C01778=1013.630,227.704,-135.004,168.137,54.282,160.252
C01779=1013.625,227.455,-134.979,168.132,54.292,160.253
C01780=1013.620,227.206,-134.953,168.128,54.302,160.254
C01781=1013.615,226.958,-134.928,168.123,54.312,160.255
C01782=1013.611,226.709,-134.903,168.118,54.322,160.256
C01783=1013.604,226.460,-134.878,168.113,54.331,160.257
C01784=1013.600,226.211,-134.853,168.109,54.341,160.258
C01785=1013.595,225.963,-134.827,168.104,54.351,160.260
C01786=1013.590,225.714,-134.803,168.099,54.361,160.261
C01787=1013.584,225.465,-134.777,168.094,54.371,160.262
C01788=1013.579,225.217,-134.753,168.090,54.381,160.263
C01789=1013.574,224.968,-134.727,168.085,54.390,160.264
C01790=1013.565,224.568,-134.687,168.077,54.407,160.266
C01791=1013.557,224.167,-134.648,168.070,54.423,160.268
C01792=1013.549,223.766,-134.607,168.062,54.439,160.269
C01793=1013.541,223.365,-134.567,168.054,54.455,160.271
C01794=1013.535,223.116,-134.543,168.050,54.466,160.272
C01795=1013.530,222.868,-134.517,168.045,54.475,160.273
C01796=1013.524,222.619,-134.492,168.040,54.485,160.274
C01797=1013.520,222.370,-134.467,168.036,54.495,160.276
C01798=1013.515,222.122,-134.442,168.031,54.506,160.277
C01799=1013.510,221.873,-134.418,168.026,54.516,160.278
C01800=1013.505,221.624,-134.393,168.021,54.526,160.279
C01801=1013.499,221.375,-134.368,168.017,54.536,160.280
C01802=1013.494,221.127,-134.343,168.012,54.546,160.281
C01803=1013.489,220.878,-134.318,168.007,54.556,160.282
C01804=1013.485,220.629,-134.294,168.003,54.566,160.283
C01805=1013.479,220.381,-134.269,167.997,54.577,160.285
C01806=1013.475,220.132,-134.244,167.993,54.587,160.286
C01807=1013.469,219.883,-134.219,167.989,54.597,160.287
C01808=1013.464,219.634,-134.194,167.984,54.607,160.288
C01809=1013.459,219.386,-134.170,167.979,54.617,160.289
C01810=1013.452,219.034,-134.135,167.973,54.632,160.291
C01811=1013.444,218.683,-134.100,167.966,54.646,160.293
C01812=1013.437,218.332,-134.066,167.959,54.661,160.294
C01813=1013.431,217.981,-134.030,167.953,54.675,160.296
C01814=1013.425,217.732,-134.006,167.949,54.686,160.297
C01815=1013.421,217.483,-133.981,167.943,54.696,160.298
C01816=1013.415,217.235,-133.957,167.939,54.706,160.299
C01817=1013.410,216.986,-133.933,167.935,54.717,160.301
C01818=1013.405,216.737,-133.908,167.929,54.727,160.302
C01819=1013.400,216.489,-133.884,167.925,54.738,160.303
C01820=1013.395,216.240,-133.859,167.920,54.748,160.304
C01821=1013.390,215.991,-133.835,167.915,54.759,160.305
C01822=1013.385,215.742,-133.811,167.911,54.770,160.307
C01823=1013.379,215.494,-133.787,167.906,54.779,160.308
C01824=1013.375,215.245,-133.762,167.901,54.790,160.309
C01825=1013.370,214.996,-133.738,167.897,54.801,160.310
C01826=1013.364,214.747,-133.714,167.892,54.811,160.311
C01827=1013.359,214.499,-133.690,167.887,54.822,160.313
C01828=1013.354,214.250,-133.666,167.883,54.833,160.314
C01829=1013.349,214.001,-133.641,167.879,54.843,160.315
C01830=1013.344,213.752,-133.617,167.873,54.854,160.316
C01831=1013.339,213.504,-133.593,167.869,54.864,160.318
C01832=1013.334,213.254,-133.569,167.864,54.875,160.319
C01833=1013.329,213.006,-133.545,167.860,54.886,160.320
C01834=1013.324,212.757,-133.520,167.855,54.896,160.321
C01835=1013.319,212.508,-133.496,167.850,54.907,160.322
C01836=1013.314,212.259,-133.472,167.846,54.918,160.324
C01837=1013.308,212.010,-133.448,167.841,54.929,160.325
C01838=1013.304,211.762,-133.423,167.837,54.939,160.326
C01839=1013.299,211.512,-133.400,167.832,54.949,160.327
C01840=1013.294,211.264,-133.376,167.827,54.960,160.329
C01841=1013.289,211.016,-133.351,167.823,54.971,160.330
C01842=1013.284,210.767,-133.328,167.818,54.982,160.331
C01843=1013.279,210.518,-133.303,167.814,54.993,160.332
C01844=1013.274,210.269,-133.279,167.809,55.003,160.334
C01845=1013.269,210.020,-133.255,167.804,55.014,160.335
C01846=1013.264,209.771,-133.231,167.800,55.024,160.336
C01847=1013.259,209.522,-133.207,167.795,55.035,160.337
C01848=1013.255,209.274,-133.183,167.791,55.046,160.339
C01849=1013.250,209.025,-133.159,167.785,55.057,160.340
C01850=1013.244,208.776,-133.135,167.781,55.068,160.341
C01851=1013.239,208.527,-133.112,167.776,55.079,160.342
C01852=1013.234,208.278,-133.087,167.772,55.090,160.344
C01853=1013.230,208.030,-133.064,167.767,55.101,160.345
C01854=1013.224,207.781,-133.040,167.763,55.111,160.346
C01855=1013.219,207.532,-133.016,167.758,55.122,160.347
C01856=1013.214,207.283,-132.993,167.754,55.133,160.349
C01857=1013.209,207.034,-132.969,167.749,55.144,160.350
C01858=1013.205,206.786,-132.945,167.745,55.156,160.352
C01859=1013.199,206.537,-132.921,167.740,55.167,160.353
C01860=1013.194,206.288,-132.898,167.735,55.178,160.354
C01861=1013.189,206.039,-132.874,167.731,55.188,160.355
C01862=1013.184,205.791,-132.851,167.726,55.200,160.357
C01863=1013.179,205.542,-132.827,167.722,55.210,160.358
C01864=1013.174,205.293,-132.804,167.717,55.221,160.359
C01865=1013.169,205.044,-132.780,167.713,55.233,160.361
C01866=1013.164,204.796,-132.756,167.708,55.244,160.362
C01867=1013.159,204.547,-132.733,167.703,55.255,160.363
C01868=1013.154,204.297,-132.709,167.699,55.266,160.365
C01869=1013.150,204.049,-132.686,167.695,55.278,160.366
C01870=1013.144,203.798,-132.662,167.690,55.289,160.367
C01871=1013.139,203.546,-132.638,167.685,55.300,160.368
C01872=1013.134,203.295,-132.616,167.681,55.311,160.370
C01873=1013.129,203.043,-132.592,167.676,55.322,160.371
C01874=1013.112,202.020,-132.502,167.137,55.220,160.221
C01875=1013.109,201.771,-132.481,167.133,55.232,160.223
C01876=1013.105,201.522,-132.458,167.127,55.245,160.224
C01877=1013.101,201.273,-132.438,167.123,55.257,160.226
C01878=1013.097,201.024,-132.415,167.119,55.269,160.227
C01879=1013.094,200.775,-132.394,167.114,55.282,160.229
C01880=1013.089,200.526,-132.372,167.109,55.294,160.230
C01881=1013.086,200.277,-132.351,167.105,55.306,160.232
C01882=1013.082,200.027,-132.329,167.100,55.318,160.233
C01883=1013.078,199.779,-132.307,167.094,55.331,160.234
C01884=1013.074,199.529,-132.286,167.090,55.343,160.236
C01885=1013.071,199.281,-132.264,167.086,55.355,160.237
C01886=1013.066,199.032,-132.242,167.082,55.368,160.239
C01887=1013.063,198.783,-132.221,167.076,55.380,160.240
C01888=1013.058,198.533,-132.200,167.072,55.393,160.242
C01889=1013.055,198.284,-132.178,167.067,55.405,160.243
C01890=1013.050,198.035,-132.157,167.063,55.417,160.245
C01891=1013.046,197.787,-132.136,167.058,55.429,160.246
C01892=1013.043,197.537,-132.114,167.053,55.442,160.247
C01893=1013.039,197.288,-132.093,167.049,55.454,160.249
C01894=1013.035,197.039,-132.073,167.044,55.467,160.250
C01895=1013.030,196.790,-132.051,167.039,55.479,160.252
C01896=1013.027,196.541,-132.030,167.035,55.492,160.253
C01897=1013.023,196.291,-132.009,167.031,55.504,160.255
C01898=1013.019,196.043,-131.988,167.025,55.517,160.256
C01899=1013.015,195.793,-131.966,167.021,55.529,160.258
C01900=1013.011,195.544,-131.946,167.017,55.541,160.259
C01901=1013.007,195.295,-131.925,167.013,55.554,160.261
C01902=1013.003,195.046,-131.904,167.007,55.566,160.262
C01903=1012.999,194.797,-131.882,167.003,55.579,160.264
C01904=1012.995,194.548,-131.861,166.998,55.591,160.265
C01905=1012.991,194.299,-131.840,166.994,55.603,160.266
C01906=1012.987,194.050,-131.820,166.990,55.615,160.268
C01907=1012.984,193.801,-131.798,166.984,55.628,160.269
C01908=1012.979,193.552,-131.777,166.980,55.640,160.271
C01909=1012.975,193.303,-131.756,166.976,55.652,160.272
C01910=1012.972,193.054,-131.735,166.972,55.665,160.274
C01911=1012.968,192.804,-131.714,166.967,55.677,160.275
C01912=1012.964,192.556,-131.693,166.963,55.690,160.277
C01913=1012.960,192.307,-131.672,166.959,55.702,160.278
C01914=1012.956,192.057,-131.650,166.955,55.714,160.280
C01915=1012.952,191.808,-131.630,166.949,55.727,160.281
C01916=1012.949,191.559,-131.610,166.945,55.739,160.282
C01917=1012.945,191.310,-131.589,166.941,55.751,160.284
C01918=1012.941,191.061,-131.567,166.936,55.763,160.285
C01919=1012.937,190.812,-131.546,166.932,55.776,160.287
C01920=1012.933,190.563,-131.525,166.928,55.788,160.288
C01921=1012.930,190.314,-131.504,166.923,55.800,160.290
C01922=1012.926,190.064,-131.484,166.919,55.813,160.291
C01923=1012.922,189.815,-131.463,166.915,55.825,160.293
C01924=1012.918,189.567,-131.442,166.911,55.837,160.294
C01925=1012.915,189.318,-131.421,166.906,55.849,160.296
C01926=1012.910,189.068,-131.400,166.902,55.861,160.297
C01927=1012.907,188.819,-131.379,166.898,55.874,160.299
C01928=1012.903,188.570,-131.359,166.893,55.886,160.300
C01929=1012.899,188.321,-131.337,166.889,55.898,160.302
C01930=1012.896,188.072,-131.317,166.885,55.911,160.303
C01931=1012.891,187.822,-131.296,166.880,55.923,160.305
C01932=1012.887,187.573,-131.275,166.876,55.935,160.306
C01933=1012.884,187.324,-131.254,166.872,55.948,160.308
C01934=1012.880,187.076,-131.233,166.867,55.960,160.309
C01935=1012.876,186.796,-131.210,166.863,55.973,160.311
C01936=1012.872,186.518,-131.186,166.858,55.987,160.312
C01937=1012.868,186.240,-131.164,166.854,56.001,160.314
C01938=1012.863,185.960,-131.140,166.849,56.014,160.315
C01939=1012.860,185.711,-131.120,166.845,56.026,160.317
C01940=1012.857,185.462,-131.099,166.840,56.038,160.319
C01941=1012.853,185.213,-131.079,166.836,56.051,160.320
C01942=1012.849,184.964,-131.058,166.832,56.063,160.322
C01943=1012.845,184.715,-131.037,166.829,56.075,160.323
C01944=1012.842,184.466,-131.016,166.824,56.087,160.324
C01945=1012.838,184.216,-130.995,166.820,56.099,160.326
C01946=1012.834,183.967,-130.974,166.816,56.112,160.328
C01947=1012.830,183.718,-130.954,166.811,56.124,160.329
C01948=1012.827,183.469,-130.933,166.807,56.136,160.330
C01949=1012.823,183.220,-130.913,166.804,56.148,160.332
C01950=1012.820,182.971,-130.892,166.799,56.160,160.333
C01951=1012.816,182.722,-130.872,166.795,56.172,160.335
C01952=1012.813,182.472,-130.851,166.791,56.184,160.336
C01953=1012.809,182.224,-130.830,166.788,56.196,160.338
C01954=1012.805,181.974,-130.810,166.783,56.208,160.339
C01955=1012.802,181.725,-130.789,166.779,56.220,160.341
C01956=1012.798,181.476,-130.768,166.774,56.232,160.342
C01957=1012.795,181.227,-130.748,166.772,56.245,160.344
C01958=1012.791,180.977,-130.728,166.767,56.257,160.345
C01959=1012.786,180.728,-130.708,166.763,56.270,160.347
C01960=1012.782,180.479,-130.688,166.759,56.282,160.348
C01961=1012.778,180.230,-130.668,166.755,56.294,160.350
C01962=1012.774,179.980,-130.648,166.751,56.307,160.351
C01963=1012.771,179.731,-130.628,166.746,56.319,160.353
C01964=1012.766,179.482,-130.609,166.742,56.331,160.354
C01965=1012.763,179.233,-130.589,166.738,56.344,160.356
C01966=1012.759,178.984,-130.569,166.735,56.355,160.357
C01967=1012.755,178.734,-130.549,166.731,56.368,160.359
C01968=1012.751,178.485,-130.529,166.727,56.380,160.360
C01969=1012.747,178.236,-130.509,166.722,56.392,160.362
C01970=1012.743,177.987,-130.489,166.719,56.405,160.363
C01971=1012.739,177.738,-130.469,166.715,56.417,160.365
C01972=1012.736,177.489,-130.449,166.711,56.429,160.366
C01973=1012.732,177.240,-130.429,166.707,56.441,160.368
C01974=1012.728,176.991,-130.410,166.703,56.454,160.369
C01975=1012.724,176.742,-130.390,166.699,56.466,160.371
C01976=1012.720,176.493,-130.370,166.695,56.478,160.372
C01977=1012.716,176.243,-130.350,166.692,56.491,160.374
C01978=1012.712,175.994,-130.331,166.687,56.503,160.375
C01979=1012.708,175.745,-130.311,166.683,56.515,160.377
C01980=1012.705,175.496,-130.291,166.680,56.527,160.378
C01981=1012.701,175.246,-130.272,166.676,56.540,160.380
C01982=1012.697,174.997,-130.252,166.672,56.552,160.382
C01983=1012.693,174.748,-130.232,166.668,56.563,160.383
C01984=1012.689,174.498,-130.212,166.664,56.576,160.384
C01985=1012.686,174.250,-130.193,166.660,56.588,160.386
C01986=1012.682,174.000,-130.173,166.657,56.600,160.388
C01987=1012.678,173.751,-130.153,166.653,56.612,160.389
C01988=1012.674,173.502,-130.134,166.649,56.624,160.391
C01989=1012.670,173.253,-130.114,166.645,56.636,160.392
C01990=1012.666,173.003,-130.094,166.641,56.648,160.394
C01991=1012.662,172.754,-130.074,166.638,56.660,160.395
C01992=1012.659,172.505,-130.055,166.634,56.673,160.397
C01993=1012.655,172.256,-130.036,166.630,56.685,160.398
C01994=1012.651,172.007,-130.016,166.627,56.697,160.400
C01995=1012.648,171.757,-129.995,166.622,56.709,160.401
C01996=1012.643,171.508,-129.976,166.619,56.721,160.403
C01997=1012.640,171.259,-129.956,166.615,56.733,160.404
C01998=1012.636,171.011,-129.937,166.611,56.745,160.406
C01999=1012.632,170.707,-129.913,166.607,56.760,160.408
C02000=1012.627,170.404,-129.889,166.602,56.775,160.409
C02001=1012.623,170.100,-129.865,166.598,56.789,160.411
C02002=1012.618,169.798,-129.841,166.593,56.804,160.413
C02003=1012.614,169.548,-129.822,166.590,56.816,160.415
C02004=1012.611,169.299,-129.802,166.586,56.828,160.416
C02005=1012.607,169.050,-129.783,166.582,56.840,160.418
C02006=1012.603,168.801,-129.763,166.578,56.852,160.419
C02007=1012.599,168.551,-129.744,166.575,56.864,160.421
C02008=1012.596,168.302,-129.724,166.571,56.876,160.422
C02009=1012.592,168.054,-129.705,166.568,56.888,160.424
C02010=1012.588,167.804,-129.685,166.565,56.899,160.425
C02011=1012.585,167.554,-129.666,166.560,56.912,160.427
C02012=1012.581,167.305,-129.646,166.557,56.923,160.428
C02013=1012.578,167.057,-129.626,166.553,56.936,160.430
C02014=1012.574,166.807,-129.608,166.550,56.947,160.431
C02015=1012.570,166.558,-129.588,166.547,56.959,160.433
C02016=1012.567,166.309,-129.568,166.543,56.971,160.434
C02017=1012.563,166.060,-129.548,166.539,56.983,160.436
C02018=1012.559,165.810,-129.529,166.536,56.995,160.437
C02019=1012.556,165.562,-129.510,166.532,57.007,160.439
C02020=1012.552,165.312,-129.491,166.529,57.019,160.440
C02021=1012.548,165.063,-129.471,166.525,57.030,160.442
C02022=1012.545,164.814,-129.451,166.521,57.042,160.443
C02023=1012.542,164.564,-129.432,166.518,57.054,160.445
C02024=1012.537,164.315,-129.413,166.515,57.066,160.446
C02025=1012.534,164.066,-129.393,166.512,57.078,160.448
C02026=1012.530,163.817,-129.374,166.508,57.090,160.449
C02027=1012.527,163.567,-129.354,166.504,57.101,160.451
C02028=1012.524,163.318,-129.335,166.501,57.113,160.452
C02029=1012.520,163.069,-129.316,166.498,57.125,160.454
C02030=1012.516,162.820,-129.296,166.494,57.137,160.455
C02031=1012.494,177.789,-130.860,166.672,56.580,160.387
C02032=1012.498,178.038,-130.880,166.675,56.568,160.386
C02033=1012.501,178.288,-130.900,166.679,56.556,160.384
C02034=1012.505,178.537,-130.920,166.683,56.543,160.383
C02035=1012.509,178.786,-130.939,166.687,56.531,160.381
C02036=1012.512,179.035,-130.959,166.692,56.519,160.380
C02037=1012.517,179.284,-130.978,166.695,56.507,160.378
C02038=1012.520,179.533,-130.998,166.699,56.494,160.377
C02039=1012.524,179.783,-131.018,166.703,56.482,160.375
C02040=1012.528,180.032,-131.038,166.707,56.470,160.374
C02041=1012.532,180.281,-131.058,166.711,56.457,160.372
C02042=1012.536,180.530,-131.078,166.715,56.445,160.371
C02043=1012.540,180.779,-131.098,166.719,56.433,160.369
C02044=1012.544,181.029,-131.118,166.722,56.421,160.368
C02045=1012.548,181.278,-131.137,166.727,56.409,160.366
C02046=1012.551,181.527,-131.157,166.731,56.396,160.365
C02047=1012.555,181.776,-131.179,166.736,56.384,160.363
C02048=1012.558,182.026,-131.199,166.739,56.373,160.362
C02049=1012.562,182.274,-131.219,166.743,56.361,160.360
C02050=1012.565,182.524,-131.240,166.747,56.348,160.359
C02051=1012.569,182.773,-131.261,166.751,56.336,160.357
C02052=1012.573,183.022,-131.281,166.756,56.323,160.356
C02053=1012.577,183.271,-131.302,166.759,56.312,160.354
C02054=1012.579,183.520,-131.322,166.763,56.300,160.353
C02055=1012.583,183.769,-131.343,166.768,56.288,160.352
C02056=1012.587,184.019,-131.363,166.772,56.275,160.350
C02057=1012.591,184.267,-131.384,166.776,56.263,160.349
C02058=1012.594,184.517,-131.405,166.779,56.251,160.347
C02059=1012.598,184.766,-131.425,166.784,56.239,160.346
C02060=1012.601,185.015,-131.445,166.788,56.227,160.344
C02061=1012.605,185.264,-131.466,166.792,56.214,160.343
C02062=1012.608,185.513,-131.487,166.796,56.202,160.341
C02063=1012.612,185.762,-131.508,166.801,56.190,160.340
C02064=1012.617,186.082,-131.534,166.806,56.175,160.338
C02065=1012.622,186.401,-131.561,166.811,56.159,160.336
C02066=1012.627,186.720,-131.587,166.817,56.143,160.334
C02067=1012.631,187.040,-131.614,166.821,56.127,160.332
C02068=1012.635,187.289,-131.635,166.826,56.115,160.331
C02069=1012.638,187.538,-131.655,166.830,56.103,160.329
C02070=1012.642,187.787,-131.676,166.834,56.091,160.328
C02071=1012.645,188.036,-131.697,166.838,56.079,160.326
C02072=1012.649,188.285,-131.717,166.843,56.067,160.325
C02073=1012.653,188.534,-131.738,166.847,56.054,160.323
C02074=1012.657,188.783,-131.759,166.851,56.042,160.322
C02075=1012.660,189.033,-131.780,166.855,56.030,160.320
C02076=1012.664,189.282,-131.801,166.860,56.018,160.319
C02077=1012.668,189.531,-131.821,166.864,56.005,160.317
C02078=1012.672,189.780,-131.842,166.868,55.993,160.316
C02079=1012.675,190.029,-131.863,166.872,55.980,160.314
C02080=1012.679,190.278,-131.884,166.877,55.968,160.313
C02081=1012.683,190.527,-131.904,166.881,55.956,160.312
C02082=1012.687,190.777,-131.925,166.885,55.943,160.310
C02083=1012.690,191.026,-131.946,166.889,55.931,160.309
C02084=1012.694,191.274,-131.967,166.895,55.919,160.307
C02085=1012.698,191.523,-131.988,166.899,55.906,160.306
C02086=1012.701,191.773,-132.008,166.903,55.894,160.304
C02087=1012.705,192.022,-132.030,166.907,55.881,160.303
C02088=1012.709,192.271,-132.050,166.912,55.869,160.301
C02089=1012.713,192.520,-132.071,166.916,55.857,160.300
C02090=1012.716,192.769,-132.093,166.920,55.845,160.298
C02091=1012.721,193.019,-132.113,166.925,55.833,160.297
C02092=1012.724,193.268,-132.134,166.930,55.820,160.295
C02093=1012.728,193.516,-132.155,166.934,55.808,160.294
C02094=1012.732,193.765,-132.176,166.938,55.795,160.292
C02095=1012.736,194.015,-132.197,166.943,55.783,160.291
C02096=1012.740,194.264,-132.218,166.947,55.771,160.290
C02097=1012.743,194.513,-132.239,166.952,55.758,160.288
C02098=1012.748,194.762,-132.260,166.957,55.746,160.287
C02099=1012.751,195.011,-132.280,166.961,55.733,160.285
C02100=1012.755,195.260,-132.301,166.965,55.721,160.284
C02101=1012.759,195.510,-132.323,166.969,55.708,160.282
C02102=1012.763,195.759,-132.344,166.975,55.696,160.281
C02103=1012.767,196.007,-132.365,166.979,55.683,160.279
C02104=1012.771,196.257,-132.386,166.983,55.671,160.278
C02105=1012.775,196.506,-132.407,166.987,55.659,160.276
C02106=1012.778,196.755,-132.428,166.993,55.646,160.275
C02107=1012.783,197.004,-132.449,166.997,55.634,160.273
C02108=1012.786,197.253,-132.470,167.002,55.622,160.272
C02109=1012.790,197.502,-132.491,167.007,55.609,160.271
C02110=1012.795,197.751,-132.512,167.011,55.597,160.269
C02111=1012.798,198.000,-132.533,167.015,55.584,160.268
C02112=1012.802,198.249,-132.554,167.020,55.571,160.266
C02113=1012.806,198.498,-132.576,167.025,55.559,160.265
C02114=1012.810,198.747,-132.596,167.029,55.546,160.263
C02115=1012.814,198.996,-132.619,167.035,55.534,160.262
C02116=1012.817,199.245,-132.640,167.039,55.522,160.261
C02117=1012.822,199.495,-132.661,167.043,55.510,160.259
C02118=1012.825,199.744,-132.683,167.048,55.498,160.258
C02119=1012.829,199.992,-132.705,167.053,55.485,160.256
C02120=1012.833,200.242,-132.726,167.057,55.473,160.255
C02121=1012.836,200.491,-132.747,167.061,55.460,160.253
C02122=1012.840,200.740,-132.770,167.067,55.448,160.252
C02123=1012.844,200.989,-132.791,167.071,55.435,160.250
C02124=1012.848,201.238,-132.812,167.076,55.423,160.249
C02125=1012.852,201.487,-132.834,167.081,55.411,160.248
C02126=1012.855,201.735,-132.855,167.086,55.398,160.246
C02127=1012.860,201.985,-132.878,167.090,55.386,160.245
C02128=1012.874,202.987,-132.965,167.632,55.486,160.396
C02129=1012.880,203.246,-132.989,167.637,55.475,160.395
C02130=1012.886,203.504,-133.013,167.643,55.463,160.393
C02131=1012.890,203.764,-133.037,167.647,55.451,160.392
C02132=1012.895,204.022,-133.061,167.652,55.439,160.391
C02133=1012.900,204.271,-133.085,167.655,55.428,160.389
C02134=1012.905,204.520,-133.108,167.661,55.417,160.388
C02135=1012.911,204.769,-133.131,167.666,55.406,160.387
C02136=1012.916,205.018,-133.155,167.669,55.395,160.385
C02137=1012.921,205.267,-133.178,167.674,55.384,160.384
C02138=1012.925,205.515,-133.202,167.679,55.372,160.383
C02139=1012.930,205.764,-133.226,167.683,55.362,160.381
C02140=1012.935,206.013,-133.249,167.688,55.351,160.380
C02141=1012.940,206.262,-133.272,167.693,55.339,160.379
C02142=1012.945,206.510,-133.297,167.697,55.329,160.378
C02143=1012.950,206.760,-133.320,167.702,55.318,160.376
C02144=1012.955,207.009,-133.344,167.706,55.307,160.375
C02145=1012.959,207.257,-133.367,167.711,55.296,160.374
C02146=1012.965,207.506,-133.391,167.716,55.285,160.373
C02147=1012.970,207.755,-133.415,167.720,55.273,160.371
C02148=1012.975,208.004,-133.438,167.725,55.262,160.370
C02149=1012.979,208.252,-133.462,167.729,55.251,160.368
C02150=1012.984,208.501,-133.486,167.734,55.240,160.367
C02151=1012.990,208.750,-133.510,167.738,55.229,160.366
C02152=1012.995,208.999,-133.533,167.743,55.219,160.365
C02153=1012.999,209.248,-133.557,167.747,55.208,160.364
C02154=1013.004,209.496,-133.581,167.753,55.197,160.362
C02155=1013.009,209.746,-133.604,167.757,55.187,160.361
C02156=1013.014,209.994,-133.629,167.762,55.175,160.360
C02157=1013.019,210.244,-133.653,167.766,55.165,160.358
C02158=1013.023,210.491,-133.677,167.771,55.154,160.357
C02159=1013.029,210.740,-133.701,167.775,55.143,160.356
C02160=1013.034,210.989,-133.724,167.780,55.133,160.355
C02161=1013.038,211.238,-133.749,167.784,55.122,160.354
C02162=1013.043,211.487,-133.773,167.790,55.111,160.352
C02163=1013.049,211.736,-133.797,167.794,55.100,160.351
C02164=1013.053,211.984,-133.820,167.799,55.089,160.350
C02165=1013.058,212.233,-133.844,167.803,55.079,160.349
C02166=1013.063,212.482,-133.869,167.808,55.068,160.348
C02167=1013.068,212.731,-133.893,167.812,55.057,160.346
C02168=1013.073,212.980,-133.917,167.816,55.047,160.345
C02169=1013.078,213.228,-133.941,167.822,55.036,160.344
C02170=1013.083,213.478,-133.966,167.826,55.026,160.343
C02171=1013.088,213.726,-133.990,167.831,55.015,160.341
C02172=1013.093,213.975,-134.014,167.835,55.004,160.340
C02173=1013.098,214.224,-134.038,167.841,54.994,160.339
C02174=1013.103,214.472,-134.061,167.845,54.983,160.338
C02175=1013.108,214.721,-134.086,167.849,54.972,160.336
C02176=1013.113,214.970,-134.111,167.854,54.961,160.335
C02177=1013.118,215.219,-134.134,167.859,54.951,160.334
C02178=1013.123,215.467,-134.158,167.864,54.940,160.333
C02179=1013.128,215.716,-134.183,167.868,54.930,160.331
C02180=1013.133,215.965,-134.207,167.873,54.920,160.330
C02181=1013.138,216.214,-134.231,167.878,54.909,160.329
C02182=1013.143,216.463,-134.255,167.883,54.899,160.328
C02183=1013.149,216.711,-134.280,167.888,54.888,160.327
C02184=1013.153,216.960,-134.304,167.892,54.877,160.326
C02185=1013.158,217.209,-134.329,167.896,54.867,160.324
C02186=1013.164,217.457,-134.353,167.902,54.856,160.323
C02187=1013.169,217.706,-134.377,167.906,54.846,160.322
C02188=1013.174,217.955,-134.402,167.910,54.835,160.321
C02189=1013.179,218.212,-134.427,167.915,54.824,160.320
C02190=1013.183,218.468,-134.453,167.920,54.814,160.319
C02191=1013.189,218.726,-134.478,167.925,54.803,160.317
C02192=1013.195,218.982,-134.503,167.930,54.792,160.316
C02193=1013.199,219.231,-134.528,167.935,54.782,160.315
C02194=1013.205,219.480,-134.552,167.939,54.772,160.314
C02195=1013.209,219.729,-134.577,167.944,54.762,160.313
C02196=1013.214,219.977,-134.601,167.949,54.752,160.312
C02197=1013.219,220.226,-134.626,167.954,54.741,160.310
C02198=1013.224,220.475,-134.652,167.958,54.731,160.309
C02199=1013.229,220.723,-134.676,167.963,54.721,160.308
C02200=1013.234,220.972,-134.701,167.967,54.711,160.307
C02201=1013.240,221.221,-134.725,167.973,54.700,160.306
C02202=1013.244,221.470,-134.750,167.977,54.690,160.305
C02203=1013.249,221.719,-134.775,167.982,54.680,160.303
C02204=1013.254,221.968,-134.799,167.986,54.670,160.302
C02205=1013.260,222.216,-134.824,167.992,54.660,160.301
C02206=1013.264,222.465,-134.849,167.997,54.650,160.300
C02207=1013.269,222.713,-134.873,168.001,54.639,160.299
C02208=1013.275,222.963,-134.899,168.005,54.629,160.298
C02209=1013.280,223.211,-134.924,168.010,54.619,160.297
C02210=1013.285,223.460,-134.948,168.016,54.609,160.296
C02211=1013.290,223.708,-134.973,168.020,54.599,160.295
C02212=1013.295,223.957,-134.998,168.025,54.589,160.293
C02213=1013.301,224.206,-135.023,168.029,54.579,160.292
C02214=1013.305,224.455,-135.048,168.034,54.569,160.291
C02215=1013.311,224.703,-135.072,168.040,54.559,160.290
C02216=1013.316,224.952,-135.098,168.044,54.548,160.289
C02217=1013.321,225.200,-135.122,168.049,54.538,160.288
C02218=1013.326,225.450,-135.147,168.053,54.528,160.287
C02219=1013.332,225.698,-135.172,168.058,54.518,160.286
C02220=1013.336,225.947,-135.197,168.063,54.509,160.285
C02221=1013.341,226.195,-135.222,168.067,54.499,160.284
C02222=1013.346,226.443,-135.247,168.072,54.489,160.282
C02223=1013.352,226.692,-135.273,168.078,54.479,160.282
C02224=1013.356,226.941,-135.297,168.083,54.469,160.280
C02225=1013.361,227.190,-135.323,168.087,54.459,160.279
C02226=1013.366,227.439,-135.348,168.092,54.449,160.278
C02227=1013.372,227.687,-135.373,168.097,54.439,160.277
C02228=1013.377,227.935,-135.399,168.101,54.429,160.276
C02229=1013.381,228.184,-135.424,168.106,54.420,160.275
C02230=1013.387,228.433,-135.450,168.111,54.410,160.274
C02231=1013.392,228.682,-135.474,168.116,54.400,160.273
C02232=1013.397,228.930,-135.499,168.120,54.390,160.272
C02233=1013.403,229.179,-135.525,168.125,54.380,160.271
C02234=1013.407,229.428,-135.550,168.130,54.370,160.270
C02235=1013.412,229.676,-135.576,168.135,54.361,160.269
C02236=1013.417,229.925,-135.602,168.140,54.351,160.268
C02237=1013.422,230.174,-135.627,168.144,54.342,160.267
C02238=1013.428,230.422,-135.652,168.149,54.332,160.266
C02239=1013.433,230.671,-135.677,168.154,54.322,160.264
C02240=1013.438,230.919,-135.703,168.159,54.313,160.264
C02241=1013.443,231.168,-135.729,168.164,54.303,160.263
C02242=1013.448,231.417,-135.754,168.169,54.293,160.261
C02243=1013.453,231.666,-135.779,168.173,54.283,160.260
C02244=1013.458,231.915,-135.805,168.179,54.274,160.260
C02245=1013.463,232.163,-135.831,168.183,54.264,160.258
C02246=1013.469,232.412,-135.857,168.188,54.255,160.257
C02247=1013.473,232.660,-135.882,168.193,54.245,160.257
C02248=1013.478,232.908,-135.908,168.198,54.236,160.255
C02249=1013.485,233.227,-135.940,168.204,54.224,160.254
C02250=1013.492,233.548,-135.974,168.211,54.211,160.253
C02251=1013.499,233.866,-136.007,168.217,54.199,160.252
C02252=1013.505,234.185,-136.039,168.223,54.187,160.250
C02253=1013.510,234.433,-136.065,168.227,54.178,160.249
C02254=1013.516,234.682,-136.090,168.232,54.168,160.248
C02255=1013.521,234.931,-136.116,168.237,54.159,160.247
C02256=1013.526,235.180,-136.142,168.242,54.149,160.246
C02257=1013.531,235.428,-136.168,168.247,54.140,160.245
C02258=1013.536,235.677,-136.193,168.252,54.130,160.244
C02259=1013.541,235.925,-136.219,168.257,54.121,160.243
C02260=1013.547,236.174,-136.245,168.262,54.111,160.242
C02261=1013.552,236.422,-136.271,168.267,54.102,160.242
C02262=1013.557,236.671,-136.296,168.272,54.092,160.240
C02263=1013.562,236.919,-136.323,168.276,54.084,160.239
C02264=1013.568,237.168,-136.349,168.281,54.074,160.238
C02265=1013.573,237.417,-136.375,168.286,54.065,160.238
C02266=1013.578,237.665,-136.400,168.291,54.055,160.236
C02267=1013.584,237.914,-136.426,168.297,54.046,160.236
C02268=1013.588,238.163,-136.452,168.301,54.036,160.235
C02269=1013.594,238.412,-136.478,168.307,54.027,160.234
C02270=1013.598,238.659,-136.505,168.311,54.018,160.233
C02271=1013.604,238.908,-136.530,168.316,54.009,160.232
C02272=1013.609,239.157,-136.556,168.321,54.000,160.231
C02273=1013.614,239.405,-136.583,168.326,53.990,160.230
C02274=1013.619,239.654,-136.609,168.331,53.982,160.229
C02275=1013.625,239.903,-136.635,168.335,53.972,160.228
C02276=1013.630,240.151,-136.661,168.341,53.963,160.227
C02277=1013.634,240.364,-136.685,168.344,53.955,160.226
C02278=1013.639,240.578,-136.706,168.349,53.947,160.226
C02279=1013.643,240.791,-136.729,168.353,53.940,160.225
C02280=1013.648,241.004,-136.752,168.358,53.932,160.224
C02281=1013.652,241.218,-136.774,168.361,53.924,160.223
C02282=1013.656,241.430,-136.797,168.366,53.916,160.222
C02283=1013.661,241.644,-136.819,168.370,53.909,160.222
C02284=1013.666,241.857,-136.842,168.375,53.901,160.221
C02285=1013.670,242.105,-136.868,168.380,53.892,160.220
C02286=1013.676,242.354,-136.895,168.384,53.883,160.219
C02287=1013.681,242.603,-136.921,168.389,53.873,160.218
C02288=1013.686,242.851,-136.947,168.394,53.864,160.217
C02289=1013.691,243.099,-136.975,168.399,53.856,160.216
C02290=1013.697,243.348,-137.001,168.404,53.847,160.216
C02291=1013.701,243.596,-137.028,168.410,53.838,160.215
C02292=1013.706,243.845,-137.055,168.414,53.830,160.214
C02293=1013.711,244.094,-137.081,168.419,53.821,160.213
C02294=1013.717,244.343,-137.108,168.425,53.812,160.212
C02295=1013.722,244.590,-137.134,168.429,53.803,160.211
C02296=1013.726,244.840,-137.161,168.434,53.794,160.210
C02297=1013.732,245.088,-137.187,168.439,53.785,160.209
C02298=1013.737,245.337,-137.215,168.444,53.776,160.208
C02299=1013.742,245.585,-137.242,168.449,53.767,160.208
C02300=1013.747,245.833,-137.268,168.454,53.759,160.207
C02301=1013.752,246.082,-137.295,168.459,53.750,160.206
C02302=1013.758,246.331,-137.321,168.465,53.741,160.205
C02303=1013.763,246.579,-137.349,168.469,53.733,160.204
C02304=1013.767,246.827,-137.375,168.474,53.724,160.203
C02305=1013.773,247.076,-137.402,168.479,53.715,160.202
C02306=1013.778,247.324,-137.429,168.484,53.706,160.202
C02307=1013.784,247.573,-137.456,168.489,53.698,160.201
C02308=1013.789,247.822,-137.483,168.494,53.689,160.200
C02309=1013.794,248.067,-137.509,168.500,53.680,160.199
C02310=1013.799,248.311,-137.535,168.504,53.672,160.198
C02311=1013.804,248.556,-137.562,168.509,53.664,160.197
C02312=1013.810,248.801,-137.589,168.514,53.655,160.197
C02313=1013.815,249.046,-137.615,168.519,53.647,160.196
C02314=1013.820,249.292,-137.642,168.524,53.638,160.195
C02315=1013.825,249.536,-137.668,168.529,53.630,160.194
C02316=1013.831,249.782,-137.695,168.534,53.621,160.193
C02317=1013.836,250.030,-137.722,168.539,53.612,160.193
C02318=1013.840,250.278,-137.749,168.545,53.604,160.192
C02319=1013.846,250.527,-137.776,168.549,53.595,160.191
C02320=1013.851,250.775,-137.803,168.554,53.586,160.190
C02321=1013.857,251.024,-137.829,168.560,53.578,160.190
C02322=1013.862,251.272,-137.857,168.564,53.569,160.189
C02323=1013.868,251.521,-137.883,168.570,53.561,160.188
C02324=1013.873,251.769,-137.911,168.575,53.553,160.187
C02325=1013.878,252.018,-137.939,168.580,53.544,160.186
C02326=1013.884,252.266,-137.965,168.585,53.536,160.185
C02327=1013.889,252.515,-137.992,168.590,53.527,160.185
C02328=1013.895,252.763,-138.019,168.595,53.519,160.184
C02329=1013.900,253.012,-138.046,168.600,53.510,160.183
C02330=1013.905,253.260,-138.074,168.605,53.502,160.182
C02331=1013.911,253.508,-138.101,168.610,53.493,160.181
C02332=1013.916,253.757,-138.129,168.615,53.485,160.181
C02333=1013.922,254.006,-138.155,168.621,53.476,160.180
C02334=1013.927,254.254,-138.182,168.627,53.468,160.179
C02335=1013.932,254.503,-138.210,168.631,53.459,160.178
C02336=1013.938,254.751,-138.237,168.637,53.451,160.178
C02337=1013.943,254.999,-138.264,168.641,53.442,160.177
C02338=1013.949,255.248,-138.291,168.647,53.434,160.176
C02339=1013.954,255.497,-138.318,168.652,53.426,160.175
C02340=1013.960,255.745,-138.346,168.657,53.417,160.174
C02341=1013.965,255.993,-138.373,168.662,53.409,160.174
C02342=1013.971,256.242,-138.400,168.667,53.400,160.173
C02343=1013.977,256.490,-138.428,168.672,53.393,160.172
C02344=1013.982,256.739,-138.455,168.678,53.384,160.172
C02345=1013.987,256.987,-138.482,168.682,53.376,160.171
C02346=1013.993,257.235,-138.510,168.688,53.368,160.170
C02347=1013.998,257.484,-138.537,168.693,53.360,160.169
C02348=1014.005,257.733,-138.564,168.699,53.351,160.169
C02349=1014.010,257.981,-138.592,168.703,53.343,160.168
C02350=1014.015,258.230,-138.619,168.709,53.335,160.167
C02351=1014.021,258.477,-138.646,168.714,53.327,160.166
C02352=1014.027,258.727,-138.674,168.720,53.318,160.165
C02353=1014.033,258.974,-138.701,168.724,53.310,160.165
C02354=1014.038,259.223,-138.729,168.729,53.302,160.164
C02355=1014.043,259.471,-138.757,168.735,53.294,160.163
C02356=1014.048,259.719,-138.785,168.740,53.286,160.163
C02357=1014.054,259.968,-138.812,168.746,53.278,160.162
C02358=1014.059,260.217,-138.840,168.751,53.270,160.161
C02359=1014.065,260.465,-138.868,168.756,53.262,160.161
C02360=1014.070,260.713,-138.896,168.761,53.254,160.160
C02361=1014.075,260.961,-138.923,168.766,53.246,160.159
C02362=1014.081,261.210,-138.952,168.771,53.238,160.159
C02363=1014.086,261.458,-138.980,168.777,53.230,160.158
C02364=1014.092,261.706,-139.008,168.782,53.222,160.157
C02365=1014.097,261.955,-139.035,168.787,53.214,160.156
C02366=1014.103,262.204,-139.063,168.793,53.206,160.156
C02367=1014.108,262.452,-139.091,168.798,53.198,160.155
C02368=1014.113,262.700,-139.119,168.802,53.190,160.154
C02369=1014.119,262.944,-139.146,168.809,53.183,160.154
C02370=1014.124,263.188,-139.174,168.814,53.175,160.153
C02371=1014.130,263.432,-139.202,168.819,53.167,160.153
C02372=1014.135,263.676,-139.229,168.823,53.159,160.152
C02373=1014.140,263.920,-139.256,168.829,53.152,160.151
C02374=1014.146,264.164,-139.285,168.834,53.144,160.151
C02375=1014.151,264.408,-139.312,168.839,53.136,160.150
C02376=1014.157,264.653,-139.340,168.845,53.129,160.149
C02377=1014.162,264.901,-139.368,168.850,53.121,160.149
C02378=1014.168,265.149,-139.396,168.855,53.113,160.148
C02379=1014.173,265.398,-139.424,168.860,53.105,160.147
C02380=1014.179,265.646,-139.452,168.866,53.098,160.147
C02381=1014.184,265.894,-139.480,168.871,53.090,160.146
C02382=1014.190,266.142,-139.510,168.876,53.082,160.145
C02383=1014.195,266.390,-139.538,168.882,53.075,160.145
C02384=1014.201,266.639,-139.566,168.887,53.067,160.144
C02385=1014.206,266.887,-139.594,168.892,53.059,160.143
C02386=1014.212,267.136,-139.622,168.898,53.052,160.143
C02387=1014.217,267.384,-139.651,168.903,53.044,160.142
C02388=1014.223,267.632,-139.680,168.908,53.037,160.142
C02389=1014.228,267.880,-139.708,168.913,53.029,160.141
C02390=1014.234,268.129,-139.736,168.920,53.021,160.141
C02391=1014.240,268.377,-139.764,168.924,53.014,160.140
C02392=1014.245,268.625,-139.794,168.929,53.006,160.139
C02393=1014.251,268.873,-139.822,168.935,52.999,160.139
C02394=1014.257,269.122,-139.850,168.940,52.992,160.138
C02395=1014.261,269.370,-139.879,168.946,52.983,160.138
C02396=1014.267,269.619,-139.908,168.951,52.976,160.137
C02397=1014.273,269.867,-139.936,168.956,52.969,160.136
C02398=1014.278,270.115,-139.965,168.962,52.961,160.136
C02399=1014.284,270.363,-139.993,168.967,52.954,160.135
C02400=1014.290,270.611,-140.022,168.973,52.946,160.135
C02401=1014.294,270.860,-140.051,168.978,52.939,160.134
C02402=1014.301,271.108,-140.080,168.983,52.931,160.134
C02403=1014.305,271.356,-140.108,168.989,52.924,160.133
C02404=1014.312,271.604,-140.137,168.994,52.917,160.133
C02405=1014.317,271.853,-140.166,169.000,52.909,160.132
C02406=1014.322,272.101,-140.195,169.005,52.902,160.131
C02407=1014.328,272.350,-140.223,169.011,52.895,160.131
C02408=1014.333,272.597,-140.253,169.016,52.888,160.130
C02409=1014.339,272.846,-140.281,169.021,52.880,160.130
C02410=1014.345,273.095,-140.311,169.026,52.873,160.129
C02411=1014.350,273.342,-140.339,169.033,52.865,160.129
C02412=1014.356,273.591,-140.368,169.038,52.858,160.128
C02413=1014.362,273.839,-140.397,169.043,52.851,160.128
C02414=1014.367,274.087,-140.426,169.049,52.844,160.127
C02415=1014.373,274.336,-140.455,169.054,52.836,160.126
C02416=1014.379,274.584,-140.484,169.059,52.829,160.126
C02417=1014.384,274.832,-140.513,169.065,52.822,160.126
C02418=1014.390,275.080,-140.542,169.071,52.815,160.125
C02419=1014.395,275.329,-140.571,169.076,52.807,160.125
C02420=1014.401,275.577,-140.600,169.082,52.800,160.124
C02421=1014.406,275.825,-140.629,169.087,52.793,160.124
C02422=1014.413,276.073,-140.658,169.092,52.786,160.123
C02423=1014.418,276.321,-140.688,169.098,52.779,160.122
C02424=1014.423,276.569,-140.717,169.103,52.772,160.122
C02425=1014.429,276.817,-140.746,169.108,52.765,160.121
C02426=1014.435,277.066,-140.776,169.115,52.757,160.121
C02427=1014.440,277.314,-140.806,169.120,52.750,160.121
C02428=1014.446,277.561,-140.834,169.126,52.743,160.120
C02429=1014.452,277.808,-140.864,169.131,52.737,160.120
C02430=1014.457,278.054,-140.893,169.137,52.730,160.119
C02431=1014.463,278.300,-140.922,169.142,52.723,160.119
C02432=1014.469,278.547,-140.951,169.148,52.716,160.118
C02433=1014.474,278.793,-140.980,169.153,52.709,160.118
C02434=1014.479,279.039,-141.009,169.159,52.702,160.117
C02435=1014.485,279.286,-141.039,169.164,52.695,160.117
C02436=1014.491,279.532,-141.068,169.170,52.688,160.116
C02437=1014.496,279.781,-141.097,169.175,52.681,160.116
C02438=1014.502,280.028,-141.128,169.181,52.675,160.116
C02439=1014.508,280.277,-141.157,169.186,52.668,160.115
C02440=1014.514,280.525,-141.186,169.192,52.661,160.115
C02441=1014.519,280.773,-141.216,169.197,52.653,160.114
C02442=1014.524,281.021,-141.245,169.203,52.647,160.114
C02443=1014.530,281.269,-141.276,169.208,52.640,160.113
C02444=1014.536,281.517,-141.305,169.214,52.633,160.113
C02445=1014.542,281.766,-141.334,169.219,52.627,160.112
C02446=1014.547,282.014,-141.364,169.225,52.620,160.112
C02447=1014.554,282.262,-141.394,169.230,52.612,160.111
C02448=1014.559,282.510,-141.423,169.236,52.606,160.111
C02449=1014.565,282.758,-141.453,169.242,52.599,160.111
C02450=1014.570,283.007,-141.483,169.248,52.592,160.110
C02451=1014.577,283.254,-141.512,169.254,52.585,160.110
C02452=1014.582,283.503,-141.542,169.260,52.579,160.110
C02453=1014.588,283.751,-141.572,169.265,52.572,160.109
C02454=1014.594,283.999,-141.601,169.270,52.565,160.109
C02455=1014.600,284.247,-141.631,169.276,52.558,160.108
C02456=1014.606,284.495,-141.661,169.282,52.552,160.108
C02457=1014.611,284.743,-141.691,169.287,52.545,160.108
C02458=1014.617,284.991,-141.721,169.293,52.539,160.107
C02459=1014.623,285.240,-141.751,169.299,52.532,160.107
C02460=1014.628,285.488,-141.781,169.305,52.525,160.106
C02461=1014.634,285.735,-141.812,169.310,52.519,160.106
C02462=1014.640,285.984,-141.841,169.316,52.512,160.106
C02463=1014.646,286.232,-141.872,169.322,52.505,160.105
C02464=1014.651,286.480,-141.901,169.328,52.499,160.105
C02465=1014.657,286.728,-141.932,169.333,52.492,160.104
C02466=1014.663,286.976,-141.962,169.339,52.486,160.104
C02467=1014.668,287.224,-141.992,169.345,52.479,160.104
C02468=1014.674,287.472,-142.022,169.350,52.472,160.103
C02469=1014.681,287.720,-142.053,169.356,52.466,160.103
C02470=1014.686,287.968,-142.083,169.362,52.460,160.103
C02471=1014.692,288.217,-142.113,169.368,52.453,160.102
C02472=1014.698,288.465,-142.143,169.373,52.447,160.102
C02473=1014.703,288.712,-142.173,169.379,52.441,160.102
C02474=1014.709,288.960,-142.204,169.385,52.434,160.101
C02475=1014.716,289.209,-142.234,169.391,52.427,160.101
C02476=1014.722,289.457,-142.265,169.396,52.421,160.101
C02477=1014.727,289.705,-142.294,169.401,52.415,160.100
C02478=1014.733,289.953,-142.325,169.407,52.409,160.100
C02479=1014.739,290.201,-142.355,169.413,52.402,160.100
C02480=1014.745,290.449,-142.386,169.419,52.396,160.099
C02481=1014.751,290.697,-142.416,169.425,52.390,160.099
C02482=1014.757,290.945,-142.447,169.431,52.383,160.099
C02483=1014.762,291.193,-142.477,169.437,52.377,160.099
C02484=1014.768,291.441,-142.508,169.442,52.371,160.098
C02485=1014.774,291.689,-142.539,169.448,52.364,160.098
C02486=1014.780,291.937,-142.569,169.454,52.358,160.098
C02487=1014.786,292.185,-142.599,169.460,52.352,160.097
C02488=1014.792,292.433,-142.630,169.466,52.345,160.097
C02489=1014.798,292.690,-142.662,169.472,52.339,160.097
C02490=1014.804,292.947,-142.695,169.478,52.333,160.097
C02491=1014.810,293.203,-142.726,169.483,52.326,160.096
C02492=1014.816,293.460,-142.758,169.489,52.320,160.096
C02493=1014.821,293.708,-142.789,169.496,52.314,160.096
C02494=1014.827,293.955,-142.820,169.501,52.308,160.096
C02495=1014.833,294.204,-142.852,169.507,52.302,160.095
C02496=1014.839,294.452,-142.882,169.513,52.295,160.095
C02497=1014.844,294.700,-142.914,169.520,52.290,160.095
C02498=1014.850,294.948,-142.944,169.525,52.283,160.095
C02499=1014.856,295.196,-142.976,169.530,52.277,160.094
C02500=1014.862,295.443,-143.006,169.537,52.272,160.094
C02501=1014.868,295.692,-143.038,169.542,52.265,160.094
C02502=1014.873,295.939,-143.069,169.549,52.260,160.094
C02503=1014.879,296.187,-143.100,169.555,52.253,160.093
C02504=1014.884,296.436,-143.132,169.561,52.248,160.093
C02505=1014.891,296.683,-143.163,169.567,52.241,160.093
C02506=1014.896,296.932,-143.194,169.572,52.235,160.093
C02507=1014.902,297.179,-143.225,169.578,52.230,160.093
C02508=1014.908,297.428,-143.257,169.584,52.223,160.092
C02509=1014.914,297.675,-143.288,169.590,52.218,160.092
C02510=1014.919,297.923,-143.319,169.596,52.212,160.092
C02511=1014.926,298.171,-143.350,169.602,52.206,160.092
C02512=1014.931,298.419,-143.382,169.608,52.200,160.091
C02513=1014.938,298.667,-143.412,169.614,52.194,160.091
C02514=1014.943,298.915,-143.444,169.620,52.189,160.091
C02515=1014.950,299.163,-143.475,169.626,52.182,160.091
C02516=1014.955,299.411,-143.506,169.632,52.177,160.091
C02517=1014.962,299.659,-143.538,169.638,52.170,160.090
C02518=1014.967,299.906,-143.569,169.644,52.165,160.090
C02519=1014.974,300.154,-143.601,169.651,52.159,160.090
C02520=1014.979,300.403,-143.632,169.656,52.153,160.090
C02521=1014.986,300.650,-143.663,169.662,52.148,160.090
C02522=1014.992,300.898,-143.695,169.668,52.142,160.090
C02523=1014.997,301.146,-143.727,169.674,52.136,160.089
C02524=1015.004,301.394,-143.758,169.680,52.130,160.089
C02525=1015.010,301.642,-143.790,169.687,52.124,160.089
C02526=1015.015,301.890,-143.821,169.693,52.119,160.089
C02527=1015.021,302.138,-143.853,169.699,52.112,160.089
C02528=1015.028,302.386,-143.884,169.704,52.107,160.089
C02529=1015.034,302.633,-143.916,169.710,52.102,160.089
C02530=1015.040,302.881,-143.947,169.717,52.096,160.088
C02531=1015.046,303.129,-143.979,169.723,52.090,160.088
C02532=1015.052,303.377,-144.010,169.729,52.085,160.088
C02533=1015.058,303.625,-144.042,169.735,52.078,160.088
C02534=1015.065,303.873,-144.074,169.742,52.073,160.088
C02535=1015.071,304.120,-144.106,169.748,52.067,160.088
C02536=1015.077,304.368,-144.137,169.753,52.062,160.088
C02537=1015.083,304.616,-144.169,169.759,52.056,160.088
C02538=1015.089,304.865,-144.201,169.766,52.051,160.087
C02539=1015.095,305.112,-144.232,169.772,52.045,160.087
C02540=1015.101,305.360,-144.264,169.778,52.039,160.087
C02541=1015.108,305.608,-144.296,169.785,52.034,160.087
C02542=1015.114,305.856,-144.328,169.791,52.028,160.087
C02543=1015.121,306.103,-144.360,169.797,52.023,160.087
C02544=1015.127,306.352,-144.392,169.804,52.017,160.087
C02545=1015.133,306.599,-144.423,169.809,52.012,160.087
C02546=1015.139,306.847,-144.455,169.815,52.006,160.087
C02547=1015.146,307.095,-144.486,169.822,52.001,160.087
C02548=1015.152,307.343,-144.519,169.828,51.995,160.086
C02549=1015.159,307.618,-144.555,169.835,51.989,160.086
C02550=1015.166,307.892,-144.589,169.842,51.982,160.086
C02551=1015.173,308.167,-144.625,169.849,51.977,160.086
C02552=1015.181,308.442,-144.660,169.856,51.971,160.086
C02553=1015.187,308.690,-144.692,169.862,51.965,160.086
C02554=1015.194,308.937,-144.724,169.869,51.960,160.086
C02555=1015.199,309.185,-144.756,169.875,51.954,160.086
C02556=1015.205,309.432,-144.789,169.882,51.949,160.086
C02557=1015.212,309.680,-144.821,169.887,51.944,160.086
C02558=1015.218,309.928,-144.853,169.893,51.938,160.086
C02559=1015.224,310.176,-144.886,169.900,51.933,160.086
C02560=1015.230,310.423,-144.919,169.906,51.928,160.086
C02561=1015.236,310.671,-144.952,169.912,51.923,160.086
C02562=1015.242,310.919,-144.984,169.918,51.917,160.086
C02563=1015.248,311.167,-145.017,169.925,51.913,160.086
C02564=1015.254,311.415,-145.050,169.931,51.907,160.086
C02565=1015.261,311.662,-145.083,169.937,51.902,160.086
C02566=1015.266,311.910,-145.116,169.944,51.897,160.086
C02567=1015.272,312.158,-145.148,169.950,51.892,160.086
C02568=1015.278,312.406,-145.181,169.957,51.887,160.086
C02569=1015.285,312.653,-145.213,169.963,51.881,160.086
C02570=1015.291,312.901,-145.246,169.969,51.877,160.086
C02571=1015.297,313.149,-145.279,169.976,51.872,160.086
C02572=1015.303,313.397,-145.312,169.982,51.866,160.086
C02573=1015.309,313.644,-145.345,169.989,51.861,160.086
C02574=1015.315,313.892,-145.378,169.995,51.857,160.086
C02575=1015.322,314.139,-145.410,170.001,51.851,160.086
C02576=1015.328,314.387,-145.443,170.008,51.846,160.086
C02577=1015.334,314.635,-145.477,170.015,51.841,160.086
C02578=1015.340,314.882,-145.509,170.021,51.836,160.086
C02579=1015.346,315.130,-145.542,170.027,51.831,160.086
C02580=1015.353,315.378,-145.575,170.033,51.826,160.086
C02581=1015.359,315.626,-145.608,170.040,51.821,160.086
C02582=1015.365,315.873,-145.642,170.047,51.816,160.086
C02583=1015.371,316.121,-145.675,170.054,51.811,160.086
C02584=1015.378,316.368,-145.707,170.059,51.806,160.086
C02585=1015.385,316.617,-145.741,170.066,51.801,160.086
C02586=1015.391,316.864,-145.773,170.073,51.796,160.086
C02587=1015.396,317.112,-145.807,170.079,51.791,160.087
C02588=1015.403,317.359,-145.840,170.086,51.787,160.087
C02589=1015.410,317.607,-145.873,170.092,51.782,160.087
C02590=1015.416,317.855,-145.906,170.099,51.777,160.087
C02591=1015.423,318.103,-145.939,170.105,51.772,160.087
C02592=1015.428,318.350,-145.973,170.112,51.767,160.087
C02593=1015.435,318.598,-146.006,170.119,51.762,160.087
C02594=1015.442,318.846,-146.039,170.126,51.757,160.087
C02595=1015.448,319.093,-146.072,170.131,51.753,160.087
C02596=1015.455,319.341,-146.105,170.138,51.748,160.087
C02597=1015.461,319.588,-146.139,170.145,51.743,160.088
C02598=1015.468,319.837,-146.172,170.152,51.738,160.088
C02599=1015.474,320.084,-146.205,170.158,51.733,160.088
C02600=1015.481,320.331,-146.239,170.165,51.728,160.088
C02601=1015.488,320.579,-146.272,170.171,51.724,160.088
C02602=1015.493,320.827,-146.306,170.178,51.719,160.088
C02603=1015.500,321.075,-146.339,170.184,51.714,160.088
C02604=1015.507,321.322,-146.372,170.192,51.710,160.088
C02605=1015.514,321.570,-146.405,170.198,51.705,160.089
C02606=1015.520,321.818,-146.439,170.205,51.700,160.089
C02607=1015.527,322.066,-146.473,170.211,51.695,160.089
C02608=1015.533,322.313,-146.506,170.218,51.690,160.089
C02609=1015.541,322.593,-146.544,170.225,51.685,160.089
C02610=1015.548,322.874,-146.582,170.233,51.680,160.089
C02611=1015.556,323.154,-146.620,170.241,51.675,160.089
C02612=1015.563,323.433,-146.658,170.249,51.669,160.090
C02613=1015.570,323.681,-146.691,170.255,51.664,160.090
C02614=1015.577,323.929,-146.725,170.263,51.660,160.090
C02615=1015.584,324.176,-146.758,170.269,51.655,160.090
C02616=1015.590,324.425,-146.792,170.275,51.651,160.090
C02617=1015.597,324.672,-146.826,170.282,51.646,160.090
C02618=1015.604,324.919,-146.859,170.289,51.642,160.091
C02619=1015.611,325.167,-146.893,170.296,51.637,160.091
C02620=1015.617,325.414,-146.927,170.303,51.632,160.091
C02621=1015.624,325.662,-146.961,170.310,51.628,160.091
C02622=1015.631,325.910,-146.994,170.317,51.623,160.091
C02623=1015.637,326.157,-147.028,170.324,51.619,160.092
C02624=1015.644,326.405,-147.063,170.330,51.615,160.092
C02625=1015.651,326.653,-147.097,170.337,51.610,160.092
C02626=1015.657,326.900,-147.131,170.344,51.606,160.092
C02627=1015.664,327.147,-147.165,170.351,51.601,160.092
C02628=1015.670,327.395,-147.199,170.358,51.597,160.093
C02629=1015.676,327.643,-147.234,170.364,51.593,160.093
C02630=1015.684,327.890,-147.268,170.371,51.588,160.093
C02631=1015.690,328.138,-147.302,170.378,51.584,160.093
C02632=1015.697,328.386,-147.337,170.386,51.580,160.094
C02633=1015.703,328.633,-147.370,170.393,51.575,160.094
C02634=1015.710,328.880,-147.405,170.400,51.571,160.094
C02635=1015.716,329.128,-147.440,170.406,51.567,160.094
C02636=1015.724,329.376,-147.474,170.413,51.562,160.095
C02637=1015.730,329.623,-147.509,170.420,51.558,160.095
C02638=1015.736,329.870,-147.543,170.427,51.554,160.095
C02639=1015.743,330.118,-147.577,170.434,51.550,160.096
C02640=1015.750,330.365,-147.612,170.442,51.545,160.096
C02641=1015.757,330.613,-147.646,170.448,51.542,160.096
C02642=1015.764,330.861,-147.681,170.455,51.537,160.097
C02643=1015.771,331.108,-147.715,170.462,51.533,160.097
C02644=1015.777,331.356,-147.750,170.469,51.528,160.097
C02645=1015.785,331.604,-147.784,170.476,51.524,160.097
C02646=1015.791,331.850,-147.819,170.483,51.520,160.098
C02647=1015.797,332.098,-147.853,170.491,51.516,160.098
C02648=1015.805,332.345,-147.888,170.498,51.512,160.098
C02649=1015.812,332.593,-147.923,170.504,51.508,160.099
C02650=1015.818,332.841,-147.957,170.511,51.504,160.099
C02651=1015.825,333.088,-147.993,170.519,51.500,160.099
C02652=1015.832,333.335,-148.028,170.526,51.495,160.100
C02653=1015.838,333.583,-148.063,170.533,51.491,160.100
C02654=1015.845,333.831,-148.097,170.540,51.488,160.100
C02655=1015.852,334.078,-148.132,170.547,51.484,160.101
C02656=1015.858,334.325,-148.168,170.554,51.480,160.101
C02657=1015.865,334.573,-148.203,170.561,51.475,160.101
C02658=1015.872,334.820,-148.238,170.569,51.472,160.102
C02659=1015.879,335.067,-148.273,170.576,51.467,160.102
C02660=1015.885,335.315,-148.308,170.583,51.463,160.102
C02661=1015.893,335.563,-148.344,170.591,51.460,160.103
C02662=1015.900,335.810,-148.379,170.598,51.455,160.103
C02663=1015.907,336.057,-148.413,170.604,51.452,160.104
C02664=1015.914,336.305,-148.448,170.612,51.448,160.104
C02665=1015.921,336.552,-148.484,170.619,51.444,160.104
C02666=1015.927,336.799,-148.519,170.626,51.440,160.105
C02667=1015.934,337.047,-148.554,170.633,51.436,160.105
C02668=1015.941,337.295,-148.589,170.641,51.432,160.106
C02669=1015.949,337.571,-148.628,170.649,51.428,160.106
C02670=1015.956,337.846,-148.668,170.657,51.423,160.107
C02671=1015.965,338.122,-148.707,170.665,51.420,160.107
C02672=1015.972,338.398,-148.747,170.673,51.415,160.107
C02673=1015.980,338.646,-148.782,170.681,51.411,160.108
C02674=1015.986,338.893,-148.817,170.688,51.407,160.108
C02675=1015.993,339.140,-148.853,170.696,51.404,160.109
C02676=1015.999,339.387,-148.889,170.703,51.400,160.109
C02677=1016.007,339.636,-148.924,170.710,51.396,160.110
C02678=1016.014,339.882,-148.960,170.718,51.392,160.110
C02679=1016.021,340.130,-148.995,170.726,51.389,160.111
C02680=1016.028,340.377,-149.032,170.732,51.385,160.111
C02681=1016.034,340.625,-149.067,170.739,51.381,160.111
C02682=1016.041,340.872,-149.103,170.747,51.378,160.112
C02683=1016.049,341.120,-149.139,170.754,51.374,160.112
C02684=1016.056,341.366,-149.174,170.762,51.371,160.113
C02685=1016.063,341.614,-149.210,170.770,51.367,160.114
C02686=1016.070,341.861,-149.246,170.777,51.363,160.114
C02687=1016.077,342.108,-149.282,170.784,51.359,160.114
C02688=1016.084,342.356,-149.318,170.792,51.356,160.115
C02689=1016.091,342.603,-149.354,170.800,51.352,160.115
C02690=1016.098,342.851,-149.390,170.807,51.349,160.116
C02691=1016.105,343.098,-149.426,170.815,51.345,160.116
C02692=1016.113,343.346,-149.462,170.822,51.341,160.117
C02693=1016.120,343.592,-149.498,170.830,51.338,160.117
C02694=1016.127,343.840,-149.534,170.838,51.334,160.118
C02695=1016.134,344.087,-149.570,170.844,51.331,160.118
C02696=1016.141,344.335,-149.606,170.852,51.327,160.119
C02697=1016.147,344.582,-149.642,170.860,51.325,160.120
C02698=1016.155,344.829,-149.678,170.867,51.321,160.120
C02699=1016.162,345.076,-149.714,170.875,51.317,160.121
C02700=1016.170,345.324,-149.751,170.883,51.314,160.121
C02701=1016.176,345.571,-149.787,170.890,51.310,160.122
C02702=1016.184,345.818,-149.823,170.898,51.307,160.122
C02703=1016.191,346.066,-149.859,170.906,51.304,160.123
C02704=1016.198,346.313,-149.896,170.913,51.300,160.124
C02705=1016.205,346.560,-149.932,170.921,51.297,160.124
C02706=1016.213,346.807,-149.968,170.929,51.293,160.125
C02707=1016.219,347.055,-150.005,170.937,51.290,160.125
C02708=1016.227,347.301,-150.042,170.944,51.287,160.126
C02709=1016.234,347.549,-150.078,170.952,51.283,160.126
C02710=1016.241,347.796,-150.114,170.960,51.280,160.127
C02711=1016.248,348.044,-150.151,170.967,51.277,160.128
C02712=1016.256,348.290,-150.188,170.975,51.274,160.128
C02713=1016.263,348.538,-150.225,170.983,51.270,160.129
C02714=1016.271,348.784,-150.261,170.991,51.267,160.130
C02715=1016.278,349.032,-150.298,170.998,51.264,160.130
C02716=1016.285,349.280,-150.334,171.006,51.261,160.131
C02717=1016.293,349.527,-150.372,171.014,51.257,160.131
C02718=1016.299,349.774,-150.408,171.022,51.254,160.132
C02719=1016.307,350.021,-150.445,171.030,51.251,160.133
C02720=1016.314,350.268,-150.482,171.038,51.248,160.133
C02721=1016.322,350.515,-150.519,171.046,51.245,160.134
C02722=1016.329,350.763,-150.556,171.054,51.241,160.135
C02723=1016.337,351.010,-150.593,171.062,51.238,160.135
C02724=1016.344,351.257,-150.630,171.070,51.235,160.136
C02725=1016.351,351.504,-150.666,171.078,51.231,160.137
C02726=1016.358,351.751,-150.704,171.086,51.228,160.137
C02727=1016.366,351.998,-150.741,171.094,51.225,160.138
C02728=1016.373,352.245,-150.778,171.102,51.223,160.139
C02729=1016.382,352.518,-150.819,171.110,51.219,160.139
C02730=1016.390,352.792,-150.860,171.119,51.215,160.140
C02731=1016.398,353.064,-150.901,171.128,51.212,160.141
C02732=1016.407,353.338,-150.942,171.137,51.209,160.142
C02733=1016.414,353.585,-150.979,171.145,51.206,160.143
C02734=1016.422,353.832,-151.016,171.153,51.203,160.143
C02735=1016.429,354.079,-151.054,171.161,51.200,160.144
C02736=1016.436,354.326,-151.091,171.169,51.197,160.145
C02737=1016.444,354.573,-151.129,171.177,51.194,160.145
C02738=1016.452,354.820,-151.166,171.185,51.191,160.146
C02739=1016.459,355.067,-151.203,171.194,51.188,160.147
C02740=1016.466,355.315,-151.241,171.202,51.185,160.148
C02741=1016.473,355.562,-151.278,171.210,51.182,160.148
C02742=1016.482,355.809,-151.316,171.218,51.179,160.149
C02743=1016.489,356.056,-151.354,171.226,51.176,160.150
C02744=1016.497,356.303,-151.391,171.234,51.173,160.151
C02745=1016.504,356.550,-151.429,171.243,51.171,160.152
C02746=1016.512,356.797,-151.466,171.252,51.168,160.152
C02747=1016.519,357.044,-151.503,171.260,51.165,160.153
C02748=1016.527,357.291,-151.542,171.268,51.162,160.154
C02749=1016.534,357.538,-151.579,171.276,51.160,160.155
C02750=1016.542,357.785,-151.617,171.284,51.157,160.155
C02751=1016.550,358.032,-151.655,171.292,51.154,160.156
C02752=1016.558,358.279,-151.692,171.302,51.151,160.157
C02753=1016.565,358.526,-151.731,171.310,51.148,160.158
C02754=1016.573,358.773,-151.768,171.318,51.145,160.159
C02755=1016.581,359.020,-151.807,171.326,51.143,160.160
C02756=1016.588,359.267,-151.844,171.334,51.140,160.160
C02757=1016.596,359.514,-151.883,171.343,51.137,160.161
C02758=1016.604,359.761,-151.921,171.351,51.134,160.162
C02759=1016.611,360.008,-151.959,171.360,51.132,160.163
C02760=1016.619,360.255,-151.997,171.368,51.129,160.164
C02761=1016.627,360.502,-152.036,171.376,51.127,160.165
C02762=1016.634,360.749,-152.073,171.386,51.124,160.166
C02763=1016.641,360.996,-152.111,171.394,51.121,160.166
C02764=1016.650,361.243,-152.150,171.402,51.119,160.167
C02765=1016.657,361.489,-152.188,171.410,51.117,160.168
C02766=1016.665,361.737,-152.227,171.419,51.113,160.169
C02767=1016.673,361.983,-152.265,171.428,51.111,160.170
C02768=1016.680,362.231,-152.304,171.436,51.109,160.171
C02769=1016.688,362.477,-152.343,171.445,51.107,160.172
C02770=1016.696,362.724,-152.381,171.454,51.103,160.173
C02771=1016.704,362.971,-152.419,171.462,51.101,160.174
C02772=1016.712,363.218,-152.458,171.470,51.099,160.175
C02773=1016.719,363.465,-152.496,171.480,51.096,160.176
C02774=1016.727,363.712,-152.535,171.488,51.094,160.177
C02775=1016.735,363.958,-152.573,171.497,51.091,160.177
C02776=1016.743,364.206,-152.612,171.505,51.089,160.178
C02777=1016.751,364.453,-152.650,171.514,51.086,160.179
C02778=1016.759,364.699,-152.689,171.523,51.084,160.180
C02779=1016.767,364.946,-152.728,171.531,51.082,160.181
C02780=1016.775,365.193,-152.766,171.540,51.079,160.182
C02781=1016.782,365.440,-152.805,171.549,51.077,160.183
C02782=1016.790,365.687,-152.844,171.558,51.074,160.184
C02783=1016.799,365.934,-152.883,171.567,51.072,160.185
C02784=1016.806,366.180,-152.921,171.575,51.070,160.186
C02785=1016.815,366.428,-152.960,171.584,51.067,160.187
C02786=1016.823,366.674,-152.999,171.593,51.065,160.188
C02787=1016.831,366.921,-153.038,171.602,51.062,160.189
C02788=1016.840,367.168,-153.077,171.611,51.060,160.190
C02789=1016.848,367.448,-153.121,171.621,51.057,160.191
C02790=1016.858,367.729,-153.166,171.631,51.055,160.192
C02791=1016.866,368.010,-153.210,171.642,51.052,160.194
C02792=1016.875,368.291,-153.256,171.651,51.050,160.195
C02793=1016.884,368.537,-153.295,171.661,51.047,160.196
C02794=1016.892,368.784,-153.335,171.669,51.045,160.197
C02795=1016.900,369.031,-153.373,171.678,51.044,160.198
C02796=1016.907,369.278,-153.413,171.687,51.041,160.199
C02797=1016.915,369.524,-153.452,171.696,51.039,160.200
C02798=1016.924,369.771,-153.492,171.706,51.037,160.201
C02799=1016.932,370.018,-153.532,171.714,51.035,160.202
C02800=1016.940,370.264,-153.571,171.724,51.032,160.203
C02801=1016.948,370.511,-153.611,171.733,51.030,160.204
C02802=1016.956,370.758,-153.650,171.742,51.028,160.206
C02803=1016.965,371.004,-153.689,171.751,51.026,160.207
C02804=1016.972,371.251,-153.729,171.761,51.024,160.208
C02805=1016.981,371.498,-153.769,171.769,51.022,160.209
C02806=1016.989,371.745,-153.809,171.779,51.020,160.210
C02807=1016.997,371.991,-153.848,171.788,51.018,160.211
C02808=1017.005,372.238,-153.888,171.797,51.016,160.212
C02809=1017.014,372.485,-153.928,171.806,51.014,160.214
C02810=1017.023,372.732,-153.968,171.816,51.012,160.215
C02811=1017.030,372.979,-154.007,171.824,51.010,160.216
C02812=1017.039,373.225,-154.047,171.834,51.008,160.217
C02813=1017.047,373.471,-154.087,171.844,51.006,160.218
C02814=1017.055,373.718,-154.127,171.853,51.004,160.219
C02815=1017.064,373.965,-154.166,171.862,51.002,160.220
C02816=1017.072,374.212,-154.207,171.871,51.000,160.222
C02817=1017.081,374.458,-154.246,171.881,50.998,160.223
C02818=1017.089,374.704,-154.287,171.891,50.996,160.224
C02819=1017.098,374.952,-154.327,171.900,50.995,160.225
C02820=1017.107,375.198,-154.367,171.909,50.993,160.226
C02821=1017.114,375.445,-154.407,171.919,50.991,160.228
C02822=1017.124,375.691,-154.447,171.928,50.989,160.229
C02823=1017.132,375.938,-154.488,171.938,50.987,160.230
C02824=1017.139,376.184,-154.528,171.948,50.985,160.231
C02825=1017.147,376.431,-154.568,171.957,50.984,160.233
C02826=1017.157,376.677,-154.609,171.967,50.982,160.234
C02827=1017.165,376.924,-154.649,171.976,50.980,160.235
C02828=1017.173,377.171,-154.690,171.986,50.978,160.236
C02829=1017.182,377.417,-154.731,171.995,50.976,160.238
C02830=1017.190,377.663,-154.771,172.005,50.974,160.239
C02831=1017.199,377.910,-154.812,172.014,50.973,160.240
C02832=1017.207,378.156,-154.853,172.024,50.971,160.241
C02833=1017.216,378.403,-154.894,172.034,50.970,160.243
C02834=1017.224,378.649,-154.934,172.044,50.968,160.244
C02835=1017.233,378.896,-154.975,172.053,50.967,160.246
C02836=1017.241,379.142,-155.015,172.063,50.965,160.247
C02837=1017.250,379.389,-155.056,172.073,50.963,160.248
C02838=1017.258,379.635,-155.096,172.083,50.961,160.249
C02839=1017.267,379.882,-155.138,172.092,50.960,160.251
C02840=1017.275,380.128,-155.179,172.102,50.959,160.252
C02841=1017.284,380.375,-155.220,172.112,50.956,160.253
C02842=1017.294,380.621,-155.261,172.122,50.955,160.255
C02843=1017.302,380.867,-155.301,172.133,50.954,160.256
C02844=1017.310,381.114,-155.342,172.142,50.951,160.258
C02845=1017.319,381.361,-155.384,172.152,50.950,160.259
C02846=1017.328,381.607,-155.424,172.162,50.949,160.260
C02847=1017.337,381.853,-155.466,172.172,50.948,160.262
C02848=1017.346,382.100,-155.507,172.182,50.946,160.263
C02849=1017.359,382.479,-155.570,172.198,50.943,160.265
C02850=1017.373,382.858,-155.633,172.212,50.941,160.267
C02851=1017.387,383.238,-155.697,172.228,50.939,160.270
C02852=1017.400,383.616,-155.761,172.244,50.937,160.272
C02853=1017.409,383.863,-155.802,172.254,50.935,160.273
C02854=1017.418,384.110,-155.843,172.265,50.934,160.275
C02855=1017.428,384.356,-155.884,172.275,50.933,160.276
C02856=1017.437,384.602,-155.926,172.285,50.931,160.278
C02857=1017.446,384.848,-155.968,172.295,50.930,160.279
C02858=1017.454,385.095,-156.010,172.305,50.928,160.281
C02859=1017.463,385.340,-156.051,172.316,50.927,160.282
C02860=1017.472,385.587,-156.093,172.326,50.926,160.284
C02861=1017.481,385.833,-156.134,172.336,50.924,160.285
C02862=1017.490,386.079,-156.176,172.347,50.923,160.286
C02863=1017.499,386.326,-156.218,172.357,50.922,160.288
C02864=1017.508,386.572,-156.260,172.367,50.921,160.290
C02865=1017.517,386.819,-156.302,172.378,50.920,160.291
C02866=1017.526,387.065,-156.344,172.388,50.918,160.293
C02867=1017.535,387.311,-156.386,172.400,50.917,160.294
C02868=1017.544,387.557,-156.428,172.410,50.916,160.296
C02869=1017.553,387.803,-156.470,172.420,50.915,160.298
C02870=1017.562,388.050,-156.512,172.431,50.913,160.299
C02871=1017.572,388.296,-156.554,172.441,50.912,160.301
C02872=1017.580,388.542,-156.596,172.452,50.911,160.302
C02873=1017.590,388.788,-156.639,172.462,50.910,160.304
C02874=1017.599,389.034,-156.682,172.474,50.909,160.305
C02875=1017.608,389.281,-156.723,172.484,50.908,160.307
C02876=1017.617,389.527,-156.766,172.494,50.906,160.308
C02877=1017.627,389.773,-156.809,172.505,50.906,160.310
C02878=1017.636,390.019,-156.850,172.515,50.905,160.312
C02879=1017.645,390.265,-156.893,172.527,50.903,160.314
C02880=1017.654,390.512,-156.936,172.538,50.903,160.315
C02881=1017.663,390.758,-156.979,172.548,50.902,160.317
C02882=1017.672,391.004,-157.020,172.559,50.901,160.319
C02883=1017.682,391.250,-157.063,172.570,50.900,160.320
C02884=1017.691,391.496,-157.105,172.581,50.899,160.322
C02885=1017.701,391.742,-157.148,172.592,50.898,160.324
C02886=1017.710,391.988,-157.191,172.603,50.897,160.325
C02887=1017.719,392.234,-157.234,172.614,50.896,160.327
C02888=1017.729,392.481,-157.277,172.624,50.895,160.329
C02889=1017.738,392.726,-157.320,172.636,50.894,160.330
C02890=1017.747,392.973,-157.363,172.647,50.893,160.332
C02891=1017.757,393.218,-157.405,172.657,50.892,160.334
C02892=1017.766,393.465,-157.448,172.669,50.891,160.336
C02893=1017.775,393.710,-157.492,172.680,50.890,160.337
C02894=1017.785,393.957,-157.535,172.691,50.890,160.339
C02895=1017.795,394.203,-157.578,172.702,50.889,160.341
C02896=1017.804,394.449,-157.621,172.713,50.888,160.343
C02897=1017.814,394.695,-157.664,172.725,50.887,160.344
C02898=1017.824,394.941,-157.708,172.735,50.886,160.346
C02899=1017.832,395.187,-157.751,172.747,50.886,160.348
C02900=1017.842,395.433,-157.794,172.758,50.885,160.350
C02901=1017.859,395.849,-157.867,172.777,50.884,160.353
C02902=1017.875,396.265,-157.941,172.796,50.883,160.356
C02903=1017.892,396.682,-158.014,172.816,50.881,160.359
C02904=1017.908,397.097,-158.088,172.835,50.880,160.362
C02905=1017.921,397.439,-158.149,172.851,50.879,160.365
C02906=1017.935,397.780,-158.210,172.867,50.878,160.367
C02907=1017.949,398.121,-158.270,172.883,50.877,160.370
C02908=1017.962,398.462,-158.331,172.899,50.877,160.373
C02909=1017.971,398.708,-158.375,172.911,50.876,160.375
C02910=1017.982,398.953,-158.418,172.923,50.875,160.377
C02911=1017.991,399.199,-158.463,172.934,50.875,160.378
C02912=1018.001,399.445,-158.507,172.946,50.874,160.380
C02913=1018.011,399.691,-158.551,172.958,50.874,160.382
C02914=1018.020,399.937,-158.595,172.969,50.874,160.384
C02915=1018.031,400.182,-158.639,172.981,50.873,160.386
C02916=1018.040,400.428,-158.683,172.993,50.873,160.388
C02917=1018.050,400.674,-158.728,173.005,50.872,160.390
C02918=1018.060,400.920,-158.771,173.017,50.872,160.392
C02919=1018.070,401.165,-158.816,173.029,50.871,160.394
C02920=1018.080,401.412,-158.861,173.041,50.871,160.396
C02921=1018.089,401.658,-158.906,173.053,50.871,160.398
C02922=1018.100,401.903,-158.950,173.065,50.870,160.400
C02923=1018.109,402.149,-158.994,173.077,50.870,160.403
C02924=1018.119,402.394,-159.039,173.088,50.870,160.404
C02925=1018.129,402.641,-159.084,173.101,50.869,160.407
C02926=1018.140,402.886,-159.128,173.113,50.869,160.409
C02927=1018.149,403.131,-159.173,173.125,50.869,160.411
C02928=1018.160,403.378,-159.218,173.137,50.868,160.413
C02929=1018.170,403.623,-159.262,173.149,50.868,160.415
C02930=1018.180,403.868,-159.307,173.162,50.868,160.417
C02931=1018.190,404.115,-159.352,173.174,50.868,160.419
C02932=1018.200,404.360,-159.397,173.186,50.867,160.421
C02933=1018.211,404.606,-159.442,173.199,50.867,160.424
C02934=1018.221,404.851,-159.487,173.211,50.867,160.426
C02935=1018.230,405.097,-159.531,173.223,50.866,160.428
C02936=1018.241,405.343,-159.577,173.236,50.866,160.430
C02937=1018.252,405.588,-159.622,173.248,50.866,160.432
C02938=1018.262,405.834,-159.667,173.261,50.866,160.434
C02939=1018.272,406.080,-159.712,173.274,50.866,160.436
C02940=1018.283,406.325,-159.757,173.286,50.866,160.439
C02941=1018.293,406.571,-159.802,173.299,50.866,160.441
C02942=1018.304,406.817,-159.848,173.311,50.866,160.443
C02943=1018.314,407.062,-159.893,173.323,50.866,160.445
C02944=1018.325,407.307,-159.938,173.337,50.865,160.448
C02945=1018.335,407.554,-159.983,173.349,50.865,160.450
C02946=1018.346,407.799,-160.029,173.362,50.865,160.452
C02947=1018.356,408.044,-160.075,173.374,50.865,160.454
C02948=1018.367,408.290,-160.119,173.388,50.865,160.456
C02949=1018.378,408.536,-160.165,173.400,50.865,160.459
C02950=1018.388,408.781,-160.211,173.413,50.865,160.461
C02951=1018.399,409.027,-160.257,173.427,50.865,160.464
C02952=1018.409,409.272,-160.303,173.439,50.865,160.466
C02953=1018.420,409.518,-160.349,173.452,50.865,160.468
C02954=1018.431,409.764,-160.395,173.466,50.865,160.471
C02955=1018.441,410.009,-160.441,173.478,50.866,160.473
C02956=1018.452,410.255,-160.487,173.491,50.866,160.475
C02957=1018.463,410.500,-160.533,173.504,50.866,160.478
C02958=1018.473,410.746,-160.578,173.517,50.866,160.480
C02959=1018.484,410.991,-160.625,173.531,50.866,160.482
C02960=1018.494,411.237,-160.672,173.544,50.866,160.485
C02961=1018.505,411.482,-160.717,173.557,50.867,160.487
C02962=1018.516,411.727,-160.764,173.570,50.867,160.490
C02963=1018.526,411.973,-160.810,173.584,50.867,160.492
C02964=1018.537,412.218,-160.857,173.597,50.867,160.495
C02965=1018.554,412.593,-160.928,173.618,50.867,160.498
C02966=1018.571,412.967,-160.998,173.638,50.867,160.502
C02967=1018.587,413.341,-161.069,173.658,50.868,160.506
C02968=1018.604,413.715,-161.140,173.679,50.868,160.509
C02969=1018.615,413.960,-161.187,173.693,50.869,160.512
C02970=1018.626,414.206,-161.233,173.707,50.869,160.515
C02971=1018.637,414.452,-161.280,173.721,50.870,160.517
C02972=1018.648,414.697,-161.327,173.734,50.870,160.520
C02973=1018.280,412.701,-161.288,173.609,50.937,160.516
C02974=1018.263,412.313,-161.215,173.588,50.936,160.512
C02975=1018.252,412.068,-161.168,173.574,50.937,160.510
C02976=1018.241,411.822,-161.122,173.560,50.937,160.508
C02977=1018.230,411.577,-161.075,173.548,50.936,160.505
C02978=1018.219,411.332,-161.029,173.534,50.936,160.503
C02979=1018.209,411.086,-160.984,173.521,50.936,160.500
C02980=1018.198,410.841,-160.937,173.507,50.936,160.498
C02981=1018.187,410.595,-160.891,173.495,50.936,160.496
C02982=1018.176,410.350,-160.845,173.481,50.936,160.493
C02983=1018.166,410.104,-160.799,173.468,50.936,160.491
C02984=1018.156,409.858,-160.753,173.455,50.936,160.488
C02985=1018.145,409.613,-160.707,173.442,50.936,160.486
C02986=1018.135,409.367,-160.661,173.429,50.936,160.484
C02987=1018.124,409.122,-160.615,173.416,50.936,160.481
C02988=1018.114,408.877,-160.569,173.403,50.937,160.479
C02989=1018.103,408.631,-160.524,173.390,50.936,160.477
C02990=1018.093,408.385,-160.478,173.378,50.936,160.475
C02991=1018.081,408.140,-160.432,173.364,50.937,160.472
C02992=1018.071,407.894,-160.387,173.351,50.936,160.470
C02993=1018.060,407.648,-160.341,173.339,50.937,160.468
C02994=1018.050,407.403,-160.297,173.326,50.937,160.466
C02995=1018.039,407.158,-160.251,173.313,50.937,160.463
C02996=1018.029,406.911,-160.206,173.301,50.937,160.461
C02997=1018.019,406.666,-160.160,173.288,50.938,160.459
C02998=1018.008,406.421,-160.116,173.275,50.938,160.457
C02999=1017.997,406.175,-160.070,173.263,50.938,160.455
C03000=1017.988,405.929,-160.025,173.250,50.938,160.452
C03001=1017.977,405.683,-159.980,173.237,50.939,160.450
C03002=1017.967,405.438,-159.936,173.225,50.939,160.448
C03003=1017.956,405.192,-159.890,173.212,50.939,160.446
C03004=1017.946,404.946,-159.845,173.200,50.939,160.444
C03005=1017.935,404.701,-159.800,173.188,50.940,160.442
C03006=1017.926,404.456,-159.756,173.176,50.940,160.439
C03007=1017.915,404.209,-159.710,173.163,50.940,160.437
C03008=1017.906,403.964,-159.665,173.150,50.942,160.435
C03009=1017.895,403.718,-159.621,173.138,50.942,160.433
C03010=1017.885,403.472,-159.576,173.126,50.942,160.431
C03011=1017.875,403.227,-159.531,173.114,50.942,160.429
C03012=1017.864,402.981,-159.487,173.101,50.943,160.427
C03013=1017.854,402.735,-159.442,173.089,50.943,160.425
C03014=1017.845,402.490,-159.397,173.077,50.943,160.423
C03015=1017.835,402.244,-159.353,173.065,50.944,160.421
C03016=1017.824,401.998,-159.308,173.053,50.945,160.419
C03017=1017.815,401.752,-159.263,173.041,50.945,160.417
C03018=1017.805,401.507,-159.219,173.029,50.945,160.415
C03019=1017.795,401.261,-159.175,173.018,50.946,160.413
C03020=1017.785,401.016,-159.130,173.005,50.946,160.411
C03021=1017.776,400.769,-159.086,172.993,50.947,160.409
C03022=1017.766,400.524,-159.041,172.981,50.948,160.407
C03023=1017.756,400.278,-158.998,172.969,50.948,160.405
C03024=1017.745,400.032,-158.953,172.957,50.949,160.403
C03025=1017.736,399.786,-158.909,172.946,50.949,160.401
C03026=1017.726,399.540,-158.865,172.934,50.950,160.399
C03027=1017.716,399.294,-158.821,172.922,50.951,160.397
C03028=1017.706,399.049,-158.777,172.910,50.951,160.395
C03029=1017.697,398.802,-158.733,172.898,50.952,160.393
C03030=1017.686,398.557,-158.689,172.887,50.952,160.391
C03031=1017.673,398.213,-158.628,172.871,50.953,160.388
C03032=1017.660,397.870,-158.566,172.855,50.954,160.386
C03033=1017.646,397.527,-158.506,172.838,50.956,160.383
C03034=1017.632,397.184,-158.445,172.823,50.956,160.381
C03035=1017.623,396.937,-158.401,172.811,50.957,160.379
C03036=1017.613,396.691,-158.358,172.799,50.958,160.377
C03037=1017.603,396.445,-158.314,172.788,50.958,160.375
C03038=1017.594,396.200,-158.271,172.777,50.960,160.373
C03039=1017.584,395.953,-158.228,172.765,50.960,160.371
C03040=1017.574,395.708,-158.184,172.754,50.961,160.370
C03041=1017.565,395.461,-158.141,172.742,50.962,160.368
C03042=1017.556,395.216,-158.098,172.730,50.963,160.366
C03043=1017.546,394.969,-158.055,172.719,50.964,160.364
C03044=1017.536,394.723,-158.011,172.708,50.965,160.362
C03045=1017.527,394.477,-157.968,172.697,50.966,160.361
C03046=1017.517,394.232,-157.925,172.685,50.966,160.359
C03047=1017.509,393.986,-157.882,172.675,50.967,160.357
C03048=1017.499,393.739,-157.839,172.663,50.969,160.355
C03049=1017.489,393.493,-157.795,172.653,50.970,160.354
C03050=1017.480,393.247,-157.752,172.641,50.971,160.352
C03051=1017.470,393.001,-157.710,172.630,50.971,160.350
C03052=1017.461,392.755,-157.667,172.618,50.972,160.348
C03053=1017.452,392.509,-157.623,172.608,50.973,160.347
C03054=1017.442,392.263,-157.581,172.597,50.974,160.345
C03055=1017.433,392.017,-157.538,172.586,50.975,160.343
C03056=1017.423,391.771,-157.495,172.575,50.976,160.342
C03057=1017.415,391.525,-157.452,172.563,50.978,160.340
C03058=1017.405,391.279,-157.410,172.553,50.979,160.338
C03059=1017.396,391.032,-157.368,172.543,50.980,160.337
C03060=1017.386,390.786,-157.325,172.531,50.981,160.335
C03061=1017.377,390.540,-157.283,172.521,50.982,160.333
C03062=1017.368,390.294,-157.240,172.510,50.983,160.332
C03063=1017.359,390.048,-157.197,172.498,50.984,160.330
C03064=1017.350,389.801,-157.155,172.488,50.986,160.329
C03065=1017.340,389.555,-157.113,172.478,50.987,160.327
C03066=1017.331,389.310,-157.070,172.466,50.988,160.325
C03067=1017.322,389.063,-157.029,172.456,50.989,160.324
C03068=1017.312,388.817,-156.986,172.445,50.990,160.322
C03069=1017.303,388.570,-156.944,172.435,50.992,160.321
C03070=1017.295,388.324,-156.901,172.424,50.993,160.319
C03071=1017.286,388.078,-156.859,172.413,50.995,160.317
C03072=1017.277,387.832,-156.817,172.403,50.995,160.316
C03073=1017.268,387.586,-156.775,172.392,50.997,160.314
C03074=1017.258,387.339,-156.733,172.382,50.998,160.313
C03075=1017.249,387.093,-156.691,172.371,51.000,160.311
C03076=1017.240,386.847,-156.649,172.361,51.001,160.310
C03077=1017.231,386.600,-156.607,172.350,51.002,160.308
C03078=1017.222,386.354,-156.565,172.340,51.003,160.307
C03079=1017.213,386.108,-156.524,172.330,51.005,160.305
C03080=1017.204,385.861,-156.482,172.319,51.006,160.303
C03081=1017.195,385.615,-156.440,172.309,51.007,160.302
C03082=1017.186,385.369,-156.398,172.299,51.009,160.301
C03083=1017.177,385.123,-156.356,172.287,51.011,160.299
C03084=1017.168,384.876,-156.314,172.277,51.012,160.298
C03085=1017.160,384.630,-156.274,172.267,51.014,160.296
C03086=1017.151,384.384,-156.233,172.257,51.015,160.295
C03087=1017.142,384.138,-156.191,172.247,51.017,160.293
C03088=1017.133,383.891,-156.149,172.236,51.018,160.292
C03089=1017.124,383.644,-156.108,172.226,51.019,160.290
C03090=1017.114,383.398,-156.067,172.216,51.021,160.289
C03091=1017.104,383.092,-156.016,172.203,51.023,160.287
C03092=1017.093,382.788,-155.964,172.190,51.025,160.285
C03093=1017.081,382.482,-155.914,172.178,51.027,160.284
C03094=1017.071,382.176,-155.863,172.166,51.029,160.282
C03095=1017.061,381.897,-155.816,172.154,51.031,160.280
C03096=1017.051,381.618,-155.770,172.143,51.033,160.279
C03097=1017.042,381.372,-155.728,172.133,51.034,160.277
C03098=1017.033,381.125,-155.687,172.123,51.036,160.276
C03099=1017.025,380.879,-155.647,172.113,51.038,160.275
C03100=1017.016,380.632,-155.606,172.103,51.039,160.273
C03101=1017.007,380.385,-155.565,172.093,51.041,160.272
C03102=1016.998,380.139,-155.525,172.083,51.043,160.271
C03103=1016.989,379.893,-155.483,172.073,51.045,160.269
C03104=1016.981,379.647,-155.442,172.064,51.046,160.268
C03105=1016.973,379.400,-155.401,172.054,51.048,160.267
C03106=1016.964,379.154,-155.361,172.044,51.049,160.265
C03107=1016.955,378.907,-155.320,172.034,51.051,160.264
C03108=1016.947,378.661,-155.279,172.024,51.053,160.263
C03109=1016.939,378.414,-155.238,172.014,51.055,160.261
C03110=1016.930,378.168,-155.198,172.004,51.057,160.260
C03111=1016.921,377.921,-155.157,171.995,51.059,160.259
C03112=1016.913,377.674,-155.117,171.985,51.060,160.258
C03113=1016.905,377.427,-155.076,171.976,51.062,160.256
C03114=1016.896,377.181,-155.036,171.966,51.064,160.255
C03115=1016.888,376.935,-154.995,171.957,51.066,160.254
C03116=1016.879,376.688,-154.954,171.947,51.067,160.253
C03117=1016.871,376.442,-154.914,171.937,51.070,160.251
C03118=1016.863,376.196,-154.873,171.927,51.072,160.250
C03119=1016.854,375.948,-154.833,171.918,51.073,160.249
C03120=1016.846,375.702,-154.793,171.909,51.075,160.248
C03121=1016.838,375.456,-154.752,171.899,51.077,160.246
C03122=1016.829,375.208,-154.712,171.889,51.080,160.245
C03123=1016.820,374.962,-154.672,171.880,51.081,160.244
C03124=1016.813,374.716,-154.632,171.870,51.083,160.243
C03125=1016.804,374.469,-154.593,171.861,51.085,160.242
C03126=1016.796,374.222,-154.552,171.852,51.087,160.240
C03127=1016.787,373.975,-154.513,171.842,51.089,160.239
C03128=1016.778,373.729,-154.473,171.833,51.092,160.238
C03129=1016.771,373.482,-154.433,171.823,51.094,160.237
C03130=1016.762,373.236,-154.393,171.814,51.096,160.236
C03131=1016.754,372.989,-154.353,171.804,51.098,160.235
C03132=1016.745,372.742,-154.313,171.795,51.100,160.234
C03133=1016.737,372.496,-154.274,171.786,51.102,160.232
C03134=1016.729,372.249,-154.234,171.776,51.104,160.231
C03135=1016.720,372.002,-154.194,171.768,51.106,160.230
C03136=1016.713,371.755,-154.155,171.758,51.108,160.229
C03137=1016.704,371.509,-154.115,171.748,51.111,160.228
C03138=1016.696,371.262,-154.076,171.740,51.113,160.227
C03139=1016.688,371.015,-154.036,171.730,51.115,160.226
C03140=1016.680,370.769,-153.997,171.722,51.117,160.225
C03141=1016.672,370.522,-153.957,171.712,51.119,160.223
C03142=1016.663,370.275,-153.917,171.702,51.122,160.222
C03143=1016.655,370.028,-153.878,171.694,51.124,160.221
C03144=1016.647,369.782,-153.838,171.684,51.126,160.220
C03145=1016.639,369.535,-153.799,171.675,51.128,160.219
C03146=1016.631,369.288,-153.759,171.666,51.131,160.218
C03147=1016.623,369.042,-153.720,171.658,51.133,160.217
C03148=1016.615,368.796,-153.681,171.648,51.135,160.216
C03149=1016.602,368.405,-153.619,171.634,51.139,160.214
C03150=1016.590,368.015,-153.556,171.619,51.143,160.213
C03151=1016.578,367.625,-153.494,171.606,51.146,160.211
C03152=1016.564,367.235,-153.432,171.592,51.150,160.210
C03153=1016.557,366.989,-153.394,171.582,51.152,160.208
C03154=1016.549,366.742,-153.354,171.574,51.155,160.207
C03155=1016.541,366.495,-153.316,171.565,51.157,160.206
C03156=1016.533,366.247,-153.277,171.556,51.160,160.206
C03157=1016.525,366.001,-153.238,171.547,51.162,160.204
C03158=1016.517,365.754,-153.199,171.538,51.165,160.204
C03159=1016.508,365.507,-153.161,171.529,51.167,160.203
C03160=1016.500,365.260,-153.122,171.521,51.170,160.202
C03161=1016.492,365.014,-153.083,171.512,51.173,160.201
C03162=1016.484,364.767,-153.045,171.503,51.175,160.200
C03163=1016.477,364.520,-153.006,171.495,51.177,160.199
C03164=1016.469,364.273,-152.968,171.485,51.180,160.198
C03165=1016.460,364.026,-152.929,171.477,51.182,160.197
C03166=1016.453,363.779,-152.891,171.468,51.185,160.196
C03167=1016.445,363.532,-152.852,171.460,51.188,160.195
C03168=1016.438,363.285,-152.813,171.450,51.191,160.194
C03169=1016.430,363.038,-152.775,171.442,51.193,160.193
C03170=1016.422,362.791,-152.737,171.433,51.195,160.192
C03171=1016.414,362.544,-152.698,171.424,51.199,160.191
C03172=1016.407,362.298,-152.660,171.416,51.201,160.191
C03173=1016.398,362.050,-152.621,171.408,51.203,160.190
C03174=1016.391,361.804,-152.583,171.399,51.207,160.189
C03175=1016.383,361.557,-152.544,171.390,51.209,160.188
C03176=1016.375,361.310,-152.506,171.382,51.212,160.187
C03177=1016.367,361.063,-152.467,171.373,51.215,160.186
C03178=1016.360,360.816,-152.430,171.365,51.217,160.185
C03179=1016.352,360.569,-152.392,171.356,51.220,160.184
C03180=1016.344,360.322,-152.353,171.347,51.223,160.184
C03181=1016.336,360.076,-152.315,171.339,51.225,160.183
C03182=1016.330,359.828,-152.277,171.331,51.228,160.182
C03183=1016.322,359.581,-152.238,171.323,51.231,160.181
C03184=1016.314,359.334,-152.200,171.314,51.234,160.180
C03185=1016.307,359.087,-152.162,171.305,51.236,160.179
C03186=1016.299,358.840,-152.124,171.297,51.239,160.179
C03187=1016.291,358.593,-152.087,171.288,51.243,160.178
C03188=1016.284,358.346,-152.049,171.280,51.245,160.177
C03189=1016.276,358.100,-152.011,171.272,51.248,160.176
C03190=1016.268,357.852,-151.973,171.264,51.251,160.175
C03191=1016.261,357.605,-151.935,171.255,51.254,160.175
C03192=1016.253,357.358,-151.898,171.247,51.257,160.174
C03193=1016.245,357.111,-151.860,171.239,51.260,160.173
C03194=1016.238,356.864,-151.823,171.231,51.262,160.172
C03195=1016.230,356.617,-151.784,171.222,51.266,160.171
C03196=1016.223,356.370,-151.747,171.214,51.268,160.171
C03197=1016.215,356.123,-151.710,171.206,51.271,160.170
C03198=1016.208,355.876,-151.672,171.198,51.274,160.169
C03199=1016.200,355.629,-151.635,171.189,51.278,160.168
C03200=1016.193,355.382,-151.597,171.181,51.281,160.168
C03201=1016.185,355.135,-151.560,171.173,51.284,160.167
C03202=1016.178,354.888,-151.523,171.165,51.286,160.166
C03203=1016.171,354.641,-151.485,171.157,51.289,160.165
C03204=1016.162,354.393,-151.448,171.148,51.293,160.165
C03205=1016.155,354.146,-151.410,171.140,51.296,160.164
C03206=1016.148,353.899,-151.373,171.132,51.299,160.163
C03207=1016.140,353.652,-151.335,171.124,51.302,160.163
C03208=1016.132,353.405,-151.298,171.116,51.305,160.162
C03209=1016.125,353.129,-151.257,171.107,51.308,160.161
C03210=1016.116,352.854,-151.216,171.097,51.313,160.160
C03211=1016.108,352.579,-151.174,171.088,51.316,160.160
C03212=1016.100,352.303,-151.133,171.079,51.319,160.159
C03213=1016.092,352.056,-151.096,171.072,51.323,160.158
C03214=1016.085,351.809,-151.059,171.064,51.326,160.157
C03215=1016.078,351.562,-151.022,171.056,51.329,160.157
C03216=1016.070,351.315,-150.985,171.047,51.333,160.156
C03217=1016.063,351.067,-150.948,171.039,51.336,160.155
C03218=1016.055,350.820,-150.911,171.032,51.339,160.155
C03219=1016.048,350.574,-150.874,171.024,51.342,160.154
C03220=1016.040,350.326,-150.838,171.016,51.346,160.154
C03221=1016.033,350.079,-150.800,171.008,51.349,160.153
C03222=1016.026,349.832,-150.764,171.001,51.352,160.152
C03223=1016.019,349.584,-150.727,170.993,51.355,160.152
C03224=1016.011,349.338,-150.691,170.984,51.359,160.151
C03225=1016.004,349.090,-150.654,170.976,51.362,160.150
C03226=1015.997,348.843,-150.616,170.968,51.366,160.150
C03227=1015.989,348.595,-150.580,170.960,51.369,160.149
C03228=1015.983,348.348,-150.544,170.953,51.372,160.148
C03229=1015.975,348.102,-150.507,170.945,51.376,160.148
C03230=1015.968,347.854,-150.470,170.937,51.379,160.147
C03231=1015.961,347.607,-150.434,170.930,51.382,160.147
C03232=1015.954,347.359,-150.397,170.922,51.386,160.146
C03233=1015.946,347.112,-150.361,170.914,51.389,160.145
C03234=1015.940,346.865,-150.324,170.906,51.392,160.145
C03235=1015.932,346.618,-150.288,170.899,51.396,160.144
C03236=1015.924,346.371,-150.252,170.890,51.400,160.144
C03237=1015.918,346.124,-150.215,170.883,51.404,160.143
C03238=1015.910,345.876,-150.179,170.875,51.407,160.143
C03239=1015.903,345.629,-150.143,170.867,51.411,160.142
C03240=1015.896,345.382,-150.106,170.859,51.414,160.141
C03241=1015.889,345.134,-150.070,170.852,51.417,160.141
C03242=1015.882,344.887,-150.035,170.844,51.421,160.140
C03243=1015.874,344.639,-149.999,170.837,51.424,160.140
C03244=1015.868,344.392,-149.962,170.829,51.428,160.139
C03245=1015.860,344.145,-149.926,170.822,51.432,160.139
C03246=1015.853,343.898,-149.890,170.814,51.435,160.138
C03247=1015.846,343.650,-149.853,170.806,51.439,160.138
C03248=1015.839,343.403,-149.818,170.799,51.443,160.138
C03249=1015.832,343.156,-149.782,170.792,51.447,160.137
C03250=1015.825,342.909,-149.746,170.784,51.450,160.136
C03251=1015.818,342.661,-149.709,170.776,51.454,160.136
C03252=1015.811,342.414,-149.674,170.769,51.457,160.135
C03253=1015.804,342.167,-149.638,170.761,51.461,160.135
C03254=1015.797,341.919,-149.603,170.754,51.465,160.134
C03255=1015.790,341.672,-149.566,170.745,51.469,160.134
C03256=1015.783,341.424,-149.530,170.738,51.473,160.133
C03257=1015.776,341.177,-149.495,170.730,51.476,160.133
C03258=1015.769,340.930,-149.459,170.723,51.480,160.132
C03259=1015.761,340.682,-149.424,170.716,51.484,160.132
C03260=1015.755,340.435,-149.387,170.708,51.488,160.132
C03261=1015.748,340.188,-149.352,170.700,51.491,160.131
C03262=1015.741,339.940,-149.317,170.693,51.496,160.131
C03263=1015.734,339.693,-149.281,170.686,51.499,160.130
C03264=1015.727,339.446,-149.246,170.679,51.503,160.130
C03265=1015.720,339.198,-149.211,170.672,51.507,160.129
C03266=1015.714,338.951,-149.174,170.664,51.510,160.129
C03267=1015.707,338.703,-149.139,170.657,51.514,160.129
C03268=1015.700,338.456,-149.103,170.649,51.518,160.128
C03269=1015.691,338.178,-149.064,170.641,51.523,160.128
C03270=1015.684,337.900,-149.024,170.633,51.527,160.127
C03271=1015.677,337.622,-148.984,170.625,51.532,160.127
C03272=1015.668,337.343,-148.945,170.617,51.536,160.126
C03273=1015.661,337.096,-148.910,170.609,51.540,160.126
C03274=1015.654,336.848,-148.875,170.602,51.544,160.126
C03275=1015.648,336.601,-148.840,170.595,51.548,160.125
C03276=1015.641,336.354,-148.805,170.587,51.552,160.125
C03277=1015.634,336.106,-148.769,170.580,51.556,160.124
C03278=1015.627,335.859,-148.734,170.573,51.561,160.124
C03279=1015.620,335.611,-148.699,170.565,51.564,160.124
C03280=1015.613,335.364,-148.664,170.558,51.568,160.123
C03281=1015.606,335.116,-148.628,170.551,51.573,160.123
C03282=1015.600,334.869,-148.593,170.544,51.577,160.123
C03283=1015.592,334.622,-148.559,170.537,51.581,160.122
C03284=1015.585,334.374,-148.524,170.529,51.585,160.122
C03285=1015.579,334.126,-148.489,170.522,51.589,160.121
C03286=1015.572,333.879,-148.454,170.515,51.593,160.121
C03287=1015.565,333.632,-148.419,170.507,51.597,160.121
C03288=1015.559,333.384,-148.384,170.500,51.602,160.121
C03289=1015.552,333.137,-148.349,170.493,51.606,160.120
C03290=1015.545,332.889,-148.314,170.486,51.610,160.120
C03291=1015.539,332.642,-148.279,170.479,51.614,160.120
C03292=1015.533,332.395,-148.244,170.472,51.619,160.119
C03293=1015.526,332.147,-148.210,170.465,51.623,160.119
C03294=1015.519,331.900,-148.175,170.458,51.627,160.119
C03295=1015.512,331.652,-148.141,170.451,51.631,160.118
C03296=1015.505,331.405,-148.106,170.444,51.635,160.118
C03297=1015.498,331.157,-148.072,170.437,51.640,160.118
C03298=1015.491,330.910,-148.037,170.430,51.644,160.117
C03299=1015.485,330.662,-148.002,170.422,51.648,160.117
C03300=1015.478,330.414,-147.969,170.416,51.653,160.117
C03301=1015.472,330.167,-147.934,170.408,51.657,160.117
C03302=1015.465,329.919,-147.899,170.401,51.662,160.116
C03303=1015.458,329.672,-147.865,170.394,51.666,160.116
C03304=1015.451,329.424,-147.831,170.387,51.670,160.116
C03305=1015.445,329.176,-147.796,170.380,51.675,160.116
C03306=1015.438,328.929,-147.763,170.373,51.679,160.115
C03307=1015.431,328.682,-147.728,170.366,51.683,160.115
C03308=1015.425,328.434,-147.693,170.359,51.688,160.115
C03309=1015.418,328.186,-147.659,170.352,51.693,160.115
C03310=1015.412,327.939,-147.625,170.346,51.696,160.114
C03311=1015.405,327.692,-147.590,170.339,51.701,160.114
C03312=1015.398,327.444,-147.556,170.332,51.706,160.114
C03313=1015.392,327.197,-147.522,170.325,51.710,160.114
C03314=1015.385,326.949,-147.488,170.318,51.715,160.113
C03315=1015.378,326.701,-147.454,170.311,51.719,160.113
C03316=1015.372,326.454,-147.420,170.304,51.724,160.113
C03317=1015.366,326.206,-147.385,170.297,51.728,160.113
C03318=1015.359,325.958,-147.352,170.290,51.733,160.113
C03319=1015.353,325.711,-147.318,170.283,51.737,160.112
C03320=1015.346,325.463,-147.284,170.276,51.742,160.112
C03321=1015.339,325.216,-147.250,170.269,51.747,160.112
C03322=1015.332,324.968,-147.217,170.262,51.752,160.112
C03323=1015.326,324.720,-147.183,170.255,51.756,160.112
C03324=1015.319,324.473,-147.149,170.250,51.761,160.112
C03325=1015.312,324.225,-147.116,170.243,51.765,160.111
C03326=1015.306,323.978,-147.083,170.236,51.770,160.111
C03327=1015.298,323.730,-147.049,170.229,51.775,160.111
C03328=1015.292,323.482,-147.015,170.222,51.780,160.111
C03329=1015.285,323.200,-146.977,170.215,51.785,160.111
C03330=1015.276,322.917,-146.938,170.207,51.791,160.111
C03331=1015.270,322.635,-146.900,170.198,51.796,160.110
C03332=1015.262,322.353,-146.862,170.191,51.802,160.110
C03333=1015.255,322.105,-146.829,170.184,51.807,160.110
C03334=1015.248,321.857,-146.795,170.178,51.811,160.110
C03335=1015.242,321.610,-146.762,170.171,51.816,160.110
C03336=1015.235,321.362,-146.728,170.164,51.821,160.110
C03337=1015.229,321.114,-146.695,170.158,51.826,160.110
C03338=1015.222,320.867,-146.662,170.151,51.831,160.109
C03339=1015.216,320.619,-146.629,170.144,51.836,160.109
C03340=1015.209,320.371,-146.596,170.137,51.841,160.109
C03341=1015.203,320.123,-146.562,170.131,51.846,160.109
C03342=1015.197,319.876,-146.529,170.124,51.850,160.109
C03343=1015.190,319.629,-146.495,170.117,51.855,160.109
C03344=1015.183,319.380,-146.462,170.110,51.860,160.109
C03345=1015.177,319.133,-146.429,170.104,51.865,160.109
C03346=1015.171,318.886,-146.395,170.097,51.870,160.109
C03347=1015.164,318.637,-146.362,170.090,51.875,160.108
C03348=1015.158,318.390,-146.330,170.085,51.880,160.109
C03349=1015.151,318.142,-146.297,170.078,51.885,160.108
C03350=1015.146,317.895,-146.263,170.071,51.890,160.108
C03351=1015.139,317.646,-146.230,170.064,51.895,160.108
C03352=1015.132,317.399,-146.197,170.058,51.900,160.108
C03353=1015.126,317.151,-146.164,170.051,51.905,160.108
C03354=1015.120,316.904,-146.131,170.045,51.911,160.108
C03355=1015.113,316.656,-146.097,170.038,51.916,160.108
C03356=1015.107,316.408,-146.064,170.031,51.920,160.108
C03357=1015.101,316.161,-146.032,170.024,51.925,160.108
C03358=1015.094,315.913,-145.999,170.019,51.931,160.108
C03359=1015.088,315.665,-145.966,170.012,51.936,160.108
C03360=1015.083,315.417,-145.933,170.006,51.941,160.108
C03361=1015.076,315.169,-145.900,169.999,51.945,160.108
C03362=1015.069,314.922,-145.867,169.993,51.951,160.108
C03363=1015.063,314.674,-145.834,169.986,51.956,160.108
C03364=1015.057,314.426,-145.801,169.979,51.962,160.108
C03365=1015.050,314.179,-145.769,169.973,51.967,160.108
C03366=1015.045,313.931,-145.735,169.966,51.972,160.107
C03367=1015.039,313.683,-145.703,169.961,51.977,160.108
C03368=1015.032,313.436,-145.670,169.954,51.982,160.107
C03369=1015.026,313.188,-145.637,169.948,51.987,160.108
C03370=1015.020,312.941,-145.604,169.941,51.992,160.107
C03371=1015.014,312.693,-145.571,169.935,51.998,160.108
C03372=1015.008,312.445,-145.538,169.928,52.003,160.107
C03373=1015.002,312.197,-145.506,169.921,52.008,160.108
C03374=1014.996,311.949,-145.474,169.916,52.013,160.108
C03375=1014.989,311.702,-145.441,169.909,52.019,160.108
C03376=1014.984,311.454,-145.407,169.903,52.024,160.107
C03377=1014.977,311.206,-145.375,169.896,52.029,160.108
C03378=1014.972,310.958,-145.343,169.890,52.034,160.107
C03379=1014.965,310.710,-145.310,169.883,52.040,160.108
C03380=1014.959,310.463,-145.277,169.877,52.045,160.107
C03381=1014.953,310.215,-145.244,169.871,52.050,160.108
C03382=1014.948,309.967,-145.212,169.865,52.056,160.108
C03383=1014.942,309.720,-145.179,169.858,52.061,160.108
C03384=1014.935,309.472,-145.147,169.852,52.066,160.108
C03385=1014.929,309.224,-145.115,169.846,52.072,160.108
C03386=1014.923,308.976,-145.082,169.839,52.077,160.108
C03387=1014.916,308.728,-145.050,169.833,52.083,160.108
C03388=1014.910,308.481,-145.019,169.827,52.089,160.108
C03389=1014.903,308.204,-144.983,169.819,52.095,160.108
C03390=1014.896,307.927,-144.948,169.812,52.101,160.108
C03391=1014.889,307.650,-144.912,169.805,52.107,160.108
C03392=1014.882,307.373,-144.876,169.799,52.113,160.108
C03393=1014.876,307.125,-144.844,169.792,52.119,160.108
C03394=1014.869,306.877,-144.813,169.786,52.124,160.109
C03395=1014.863,306.629,-144.781,169.780,52.130,160.109
C03396=1014.857,306.382,-144.750,169.774,52.135,160.109
C03397=1014.851,306.134,-144.717,169.768,52.142,160.109
C03398=1014.844,305.886,-144.686,169.761,52.147,160.109
C03399=1014.838,305.638,-144.653,169.755,52.153,160.109
C03400=1014.831,305.390,-144.622,169.749,52.159,160.109
C03401=1014.826,305.143,-144.590,169.742,52.164,160.109
C03402=1014.820,304.895,-144.558,169.736,52.170,160.109
C03403=1014.813,304.647,-144.527,169.730,52.176,160.110
C03404=1014.807,304.398,-144.495,169.724,52.181,160.110
C03405=1014.801,304.151,-144.464,169.718,52.188,160.110
C03406=1014.795,303.903,-144.432,169.711,52.193,160.110
C03407=1014.788,303.655,-144.400,169.705,52.199,160.110
C03408=1014.783,303.408,-144.369,169.699,52.204,160.110
C03409=1014.776,303.160,-144.337,169.693,52.211,160.111
C03410=1014.770,302.911,-144.305,169.687,52.216,160.111
C03411=1014.764,302.664,-144.274,169.680,52.222,160.111
C03412=1014.759,302.415,-144.243,169.674,52.228,160.111
C03413=1014.752,302.168,-144.211,169.668,52.234,160.111
C03414=1014.746,301.920,-144.180,169.662,52.240,160.111
C03415=1014.740,301.672,-144.148,169.655,52.245,160.111
C03416=1014.734,301.425,-144.117,169.650,52.252,160.112
C03417=1014.728,301.176,-144.085,169.643,52.257,160.112
C03418=1014.722,300.928,-144.054,169.637,52.264,160.112
C03419=1014.717,300.680,-144.022,169.631,52.269,160.112
C03420=1014.710,300.432,-143.991,169.625,52.275,160.112
C03421=1014.704,300.185,-143.959,169.620,52.281,160.113
C03422=1014.698,299.936,-143.928,169.614,52.286,160.113
C03423=1014.693,299.689,-143.897,169.608,52.293,160.113
C03424=1014.686,299.441,-143.865,169.602,52.298,160.113
C03425=1014.681,299.193,-143.834,169.596,52.305,160.113
C03426=1014.674,298.945,-143.803,169.589,52.310,160.113
C03427=1014.669,298.697,-143.771,169.583,52.317,160.114
C03428=1014.662,298.449,-143.741,169.577,52.322,160.114
C03429=1014.657,298.201,-143.709,169.571,52.329,160.114
C03430=1014.650,297.953,-143.678,169.565,52.334,160.114
C03431=1014.645,297.705,-143.647,169.559,52.341,160.114
C03432=1014.639,297.458,-143.616,169.553,52.346,160.115
C03433=1014.633,297.209,-143.584,169.547,52.353,160.115
C03434=1014.628,296.961,-143.553,169.541,52.359,160.115
C03435=1014.621,296.713,-143.522,169.535,52.365,160.115
C03436=1014.616,296.465,-143.491,169.529,52.371,160.116
C03437=1014.610,296.218,-143.460,169.523,52.377,160.116
C03438=1014.605,295.969,-143.429,169.517,52.383,160.116
C03439=1014.598,295.722,-143.397,169.511,52.389,160.116
C03440=1014.593,295.474,-143.366,169.505,52.396,160.117
C03441=1014.587,295.226,-143.335,169.500,52.401,160.117
C03442=1014.582,294.978,-143.304,169.494,52.407,160.117
C03443=1014.576,294.730,-143.274,169.488,52.414,160.117
C03444=1014.570,294.482,-143.242,169.482,52.420,160.118
C03445=1014.564,294.234,-143.211,169.476,52.426,160.118
C03446=1014.559,293.986,-143.180,169.470,52.432,160.118
C03447=1014.553,293.739,-143.149,169.464,52.438,160.118
C03448=1014.547,293.490,-143.118,169.458,52.445,160.119
C03449=1014.541,293.231,-143.087,169.453,52.451,160.119
C03450=1014.535,292.972,-143.054,169.446,52.458,160.119
C03451=1014.530,292.713,-143.021,169.440,52.464,160.119
C03452=1014.524,292.455,-142.989,169.434,52.471,160.120
C03453=1014.517,292.206,-142.959,169.428,52.477,160.120
C03454=1014.511,291.958,-142.928,169.422,52.483,160.120
C03455=1014.506,291.710,-142.897,169.416,52.490,160.121
C03456=1014.500,291.462,-142.867,169.411,52.496,160.121
C03457=1014.494,291.214,-142.836,169.405,52.502,160.121
C03458=1014.488,290.966,-142.806,169.399,52.509,160.121
C03459=1014.482,290.718,-142.775,169.393,52.515,160.122
C03460=1014.477,290.470,-142.745,169.387,52.523,160.122
C03461=1014.471,290.222,-142.715,169.381,52.529,160.122
C03462=1014.465,289.974,-142.685,169.375,52.535,160.123
C03463=1014.459,289.726,-142.654,169.369,52.542,160.123
C03464=1014.453,289.478,-142.624,169.363,52.548,160.123
C03465=1014.448,289.230,-142.593,169.357,52.554,160.124
C03466=1014.442,288.982,-142.563,169.352,52.561,160.124
C03467=1014.437,288.733,-142.533,169.346,52.568,160.124
C03468=1014.430,288.485,-142.502,169.340,52.574,160.125
C03469=1014.424,288.237,-142.472,169.335,52.581,160.125
C03470=1014.418,287.989,-142.442,169.329,52.588,160.126
C03471=1014.413,287.741,-142.412,169.323,52.594,160.126
C03472=1014.407,287.493,-142.382,169.317,52.600,160.126
C03473=1014.401,287.245,-142.351,169.312,52.607,160.127
C03474=1014.396,286.997,-142.322,169.306,52.614,160.127
C03475=1014.390,286.749,-142.291,169.300,52.620,160.127
C03476=1014.384,286.501,-142.261,169.294,52.628,160.128
C03477=1014.379,286.253,-142.231,169.288,52.634,160.128
C03478=1014.373,286.005,-142.201,169.283,52.641,160.128
C03479=1014.367,285.756,-142.171,169.277,52.647,160.129
C03480=1014.362,285.509,-142.141,169.271,52.654,160.129
C03481=1014.355,285.260,-142.112,169.266,52.661,160.130
C03482=1014.349,285.013,-142.082,169.260,52.667,160.130
C03483=1014.344,284.764,-142.052,169.254,52.674,160.130
C03484=1014.338,284.516,-142.022,169.249,52.681,160.131
C03485=1014.333,284.268,-141.992,169.243,52.688,160.131
C03486=1014.327,284.020,-141.962,169.237,52.694,160.131
C03487=1014.321,283.772,-141.932,169.231,52.702,160.132
C03488=1014.315,283.524,-141.903,169.226,52.709,160.132
C03489=1014.309,283.276,-141.873,169.220,52.715,160.133
C03490=1014.304,283.027,-141.843,169.214,52.722,160.133
C03491=1014.298,282.779,-141.813,169.209,52.729,160.134
C03492=1014.292,282.531,-141.784,169.203,52.736,160.134
C03493=1014.286,282.283,-141.754,169.198,52.743,160.135
C03494=1014.281,282.034,-141.724,169.191,52.750,160.135
C03495=1014.274,281.786,-141.695,169.186,52.757,160.135
C03496=1014.269,281.539,-141.666,169.180,52.764,160.136
C03497=1014.264,281.290,-141.636,169.175,52.771,160.136
C03498=1014.258,281.042,-141.606,169.170,52.778,160.137
C03499=1014.252,280.794,-141.577,169.164,52.785,160.137
C03500=1014.246,280.546,-141.547,169.158,52.791,160.138
C03501=1014.241,280.297,-141.518,169.152,52.799,160.138
C03502=1014.235,280.049,-141.488,169.147,52.806,160.138
C03503=1014.230,279.801,-141.459,169.141,52.813,160.139
C03504=1014.224,279.553,-141.430,169.136,52.820,160.140
C03505=1014.218,279.306,-141.400,169.130,52.826,160.140
C03506=1014.213,279.058,-141.371,169.125,52.833,160.140
C03507=1014.207,278.811,-141.341,169.119,52.840,160.141
C03508=1014.202,278.563,-141.312,169.113,52.848,160.141
C03509=1014.196,278.316,-141.283,169.108,52.855,160.142
C03510=1014.190,278.069,-141.254,169.102,52.862,160.142
C03511=1014.185,277.821,-141.225,169.097,52.869,160.143
C03512=1014.179,277.574,-141.195,169.091,52.876,160.143
C03513=1014.174,277.326,-141.166,169.086,52.883,160.144
C03514=1014.168,277.078,-141.136,169.081,52.891,160.144
C03515=1014.162,276.829,-141.107,169.074,52.898,160.145
C03516=1014.158,276.581,-141.079,169.069,52.905,160.145
C03517=1014.152,276.333,-141.049,169.064,52.912,160.146
C03518=1014.146,276.084,-141.019,169.058,52.919,160.146
C03519=1014.141,275.837,-140.991,169.053,52.926,160.147
C03520=1014.135,275.588,-140.961,169.047,52.934,160.147
C03521=1014.129,275.340,-140.932,169.041,52.941,160.148
C03522=1014.124,275.092,-140.904,169.036,52.948,160.148
C03523=1014.118,274.844,-140.874,169.030,52.955,160.149
C03524=1014.112,274.596,-140.845,169.026,52.963,160.149
C03525=1014.107,274.347,-140.817,169.019,52.971,160.150
C03526=1014.101,274.099,-140.788,169.014,52.978,160.150
C03527=1014.096,273.850,-140.759,169.009,52.985,160.151
C03528=1014.090,273.603,-140.730,169.003,52.992,160.151
C03529=1014.085,273.354,-140.700,168.997,53.000,160.152
C03530=1014.079,273.106,-140.673,168.992,53.007,160.152
C03531=1014.074,272.858,-140.643,168.987,53.014,160.153
C03532=1014.068,272.609,-140.615,168.982,53.022,160.154
C03533=1014.063,272.361,-140.585,168.975,53.030,160.154
C03534=1014.057,272.112,-140.557,168.970,53.037,160.155
C03535=1014.051,271.865,-140.528,168.965,53.045,160.155
C03536=1014.046,271.616,-140.499,168.960,53.052,160.156
C03537=1014.041,271.369,-140.471,168.953,53.059,160.156
C03538=1014.035,271.119,-140.442,168.949,53.067,160.157
C03539=1014.029,270.871,-140.413,168.943,53.074,160.157
C03540=1014.024,270.623,-140.385,168.937,53.082,160.158
C03541=1014.018,270.375,-140.355,168.932,53.089,160.159
C03542=1014.013,270.127,-140.327,168.927,53.097,160.159
C03543=1014.007,269.878,-140.299,168.922,53.104,160.160
C03544=1014.002,269.630,-140.270,168.915,53.112,160.160
C03545=1013.996,269.382,-140.241,168.910,53.120,160.161
C03546=1013.991,269.133,-140.213,168.905,53.127,160.161
C03547=1013.986,268.886,-140.184,168.899,53.135,160.162
C03548=1013.980,268.637,-140.156,168.894,53.142,160.163
C03549=1013.975,268.389,-140.128,168.889,53.150,160.163
C03550=1013.969,268.140,-140.099,168.884,53.158,160.164
C03551=1013.964,267.892,-140.071,168.878,53.165,160.164
C03552=1013.958,267.644,-140.042,168.873,53.173,160.165
C03553=1013.952,267.396,-140.014,168.868,53.181,160.166
C03554=1013.947,267.147,-139.986,168.862,53.189,160.166
C03555=1013.942,266.899,-139.957,168.857,53.196,160.167
C03556=1013.937,266.650,-139.929,168.851,53.205,160.168
C03557=1013.931,266.402,-139.901,168.846,53.212,160.168
C03558=1013.925,266.154,-139.873,168.841,53.220,160.169
C03559=1013.919,265.905,-139.844,168.835,53.228,160.170
C03560=1013.914,265.657,-139.816,168.830,53.236,160.170
C03561=1013.909,265.409,-139.788,168.825,53.243,160.171
C03562=1013.903,265.160,-139.760,168.819,53.251,160.171
